	extAprSw					:BOOL:=FALSE;//气缸伸出感应器信号,需要链接到实际的IO点
	retAprSw					:BOOL:=FALSE;//气缸收回感应器信号,需要链接到实际的IO点
	enableExtAprSw				:BOOL:=TRUE;//启用伸出感应器,针对只有一个传感器的气缸
	enableRetAprSw				:BOOL:=TRUE;//启用收回感应器,针对只有一个传感器的气缸
	noteWTXT_Ext				:WSTRING(255):="";//气缸伸出动作NoteTXT 中文
	noteWTXT_Ret				:WSTRING(255):="";//气缸缩回动作NoteTXT 中文
END_VAR
VAR_OUTPUT
	extRelay				:BOOL:=FALSE;//气缸伸出执行继电器,需要链接到实际的IO点
	retRelay				:BOOL:=FALSE;//气缸收回执行继电器,需要链接到实际的IO点
	note_Ext				:BOOL:=FALSE;// 操作提示：true 伸出、打开执行无法下发
	note_Ret				:BOOL:=FALSE;// 操作提示：true 缩回、关闭执行无法下发
	busy					:BOOL;//气缸动作Busy状态
	done					:BOOL;//气缸动作Done状态
	extdone					:BOOL;//气缸动作伸出完成
	retdone					:BOOL;//气缸动作收回完成
	error					:BOOL;//气缸动作error状态
	errID					:UDINT;//气缸动作errID
	errTXT					:STRING(255):='';//气缸动作errTXT
	errWTXT					:WSTRING(255):="";//气缸动作errTXT 中文
	sensorShow				:STRING;
END_VAR
	
VAR
	firstPower:BOOL:=TRUE;
	extErrorDelayTon		:Ton;
	extDoneDelayTon			:Ton;
	retErrorDelayTon		:Ton;
	retDoneDelayTon			:Ton;
	
	extendTrigRAlc			:R_Trig;//上升沿触发
	
	singleControlR			:R_Trig;//上升沿触发
	singleControlF			:F_Trig;//上升沿触发
	
	extendTrigR1			:R_Trig;//上升沿触发
	retractTrigR1			:R_Trig;//上升沿触发
	resetTrigR1				:R_Trig;//上升沿触发
	stopTrigR1				:R_Trig;//上升沿触发
	powerTrigR1				:R_Trig;//上升沿触发
	
	errorStep				:UINT:=0;
	
	notBusyMonitorDelayTon:TON;//动作不切换时，延迟检测
	notBusyMonitorDelayTime:TIME:=T#2S;//动作不切换延迟检测时间
	noteTON_P:tON;            // 操作提示标志位延时继电器
	noteTON_N:tON;            // 操作提示标志位延时继电器
	noteRTrig_P:R_TRIG;          // 操作提示
	noteRTrig_N:R_TRIG;          // 操作提示
	extcheckDelayTime	:TON; // 输出到输入检测时间
	extcheckDelayTimeS	:TIME; // 输出到输入检测时间
	extcheckRtrig:R_TRIG;     // 输出到输入检测
	retcheckDelayTime	:TON; // 输出到输入检测时间
	retcheckDelayTimeS	:TIME; // 输出到输入检测时间
	retcheckRtrig:R_TRIG;     // 输出到输入检测
	extRealayRtrig:R_TRIG;
	retRealayRtrig:R_TRIG;
END_VAR

// 实时读取设置的流量值以及实际反馈浏览值
// ****************************
Init_ACT();
Error_ACT();
Extend_ACT();
Retract_ACT();
Reset_ACT();
Error_ACT();
SafeMonitor_ACT();
//首次上电，传感器状态决定电磁阀输出信号
//IF NOT firstPower THEN
//	IF extAprSw AND NOT retAprSw THEN
//		extend:=TRUE;
//		firstPower:=TRUE;
//	END_IF
//	IF retAprSw AND NOT extAprSw THEN
//		retract:=TRUE;
//		firstPower:=TRUE;
//	END_IF
//	IF (NOT extAprSw) AND (NOT retAprSw) THEN
//		errorStep:=3;
//	END_IF
//	IF (extAprSw) AND (retAprSw) THEN
//		errorStep:=3;
//	END_IF
//END_IF

(*
触发伸出动作，成功触发返回TRUE，触发失败返回FALSE
*)
METHOD Act_Extend : BOOL
VAR_INPUT
END_VAR
IF enable AND extCondition THEN// AND NOT busy
	Act_Extend:=extend:=TRUE;
ELSE
	Act_Extend:=FALSE;
END_IF
END_METHOD

(*
触发复位报警动作，成功触发返回TRUE，触发失败返回FALSE
*)
METHOD Act_Reset : BOOL
VAR_INPUT
END_VAR
Act_Reset:=reset:=TRUE;
END_METHOD

(*
触发缩回动作，成功触发返回TRUE，触发失败返回FALSE
*)
METHOD Act_Retract : BOOL
VAR_INPUT
END_VAR
IF enable AND retCondition THEN// AND NOT busy
	Act_Retract:=retract:=TRUE;
ELSE
	Act_Retract:=FALSE;
END_IF
END_METHOD

(*
触发停止输出动作，成功触发返回TRUE，触发失败返回FALSE
*)
METHOD Act_Stop : BOOL
VAR_INPUT
END_VAR
Act_Stop:=stop:=TRUE;
END_METHOD

ACTION Error_ACT:
CASE errorStep OF
	0:
		error:=FALSE;
		errID:=0;
		errTXT:='';
 (*
	1:
		error:=TRUE;
		errID:=errorID+errorStep;
		errTXT:=CONCAT(STR1:=nameTXT,STR2:=' Extend Error!');
		errWTXT:=WCONCAT(STR1:=TO_WSTRING(nameTXT),STR2:=" 伸出(打开)错误");
	2:
		error:=TRUE;
		errID:=errorID+errorStep;
		errTXT:=CONCAT(STR1:=nameTXT,STR2:=' Retract Error!');
		errWTXT:=WCONCAT(STR1:=TO_WSTRING(nameTXT),STR2:=" 缩回(关闭)错误");
		*)
	1..3:
		error:=TRUE;
		errID:=getErrID(errorStep);
		errTXT:=getErrTXT(errorStep);
		errWTXT:=getErrWTXT(errorStep);
END_CASE
END_ACTION

ACTION Extend_ACT:
//气缸伸出--extend 触发
IF extend AND NOT extCondition THEN
	note_Ext:=TRUE;
	note_Ret:=FALSE;
	NoteHMI.showFlag:=TRUE;
	NoteHMI.showText:='';
	NoteHMI.showText:=CONCAT(NoteHMI.showText,nameTXT);
	NoteHMI.showText:=CONCAT(NoteHMI.showText,' Ext Condition Not Satisfied!');
	operatorLog.append(CONCAT(nameTXT,' Extend Not Done'));
END_IF
IF extend AND enable AND extCondition THEN// AND NOT busy
	busy:=TRUE;
	retract:=FALSE;
	extdone:=FALSE;
	retdone:=FALSE;
	extStep:=10;
	retStep:=0;
	note_Ext:=FALSE;
	note_Ret:=FALSE;
	operatorLog.append(CONCAT(nameTXT,' Extend Done'));
	//errorStep:=0;
END_IF
extend:=FALSE;
extcheckDelayTime(IN:=extStep>10 AND NOT extcheckRtrig.Q,PT:=T#60S);
extcheckRtrig(CLK:=extAprSw);
IF extcheckRtrig.Q THEN
	extcheckDelayTimeS:=extcheckDelayTime.ET;
END_IF
CASE extStep OF
0:
	//ready
10:
	firstPower:=FALSE;
	extErrorDelayTon(IN:=FALSE);
	extDoneDelayTon(IN:=FALSE);
	extStep:=20;
	extRelay:=TRUE;
	retRelay:=FALSE;
20:
	extErrorDelayTon(IN:=(NOT extAprSw AND enableExtAprSw),PT:=errorDelayTime);
	IF extErrorDelayTon.Q THEN
		//done:=FALSE;
		extdone:=FALSE;
		retdone:=FALSE;
		errorStep:=1;
		RETURN;
	END_IF
	IF enableExtAprSw THEN
		extDoneDelayTon(IN:=extAprSw,PT:=doneDelayTimeShortExtend);
	ELSE
		extDoneDelayTon(IN:=NOT enableExtAprSw,PT:=doneDelayTimeLongExtend);
	END_IF
	
	IF extDoneDelayTon.Q THEN
		IF NOT retAprSw THEN
			busy:=FALSE;
			//done:=TRUE;
			extdone:=TRUE;
			retdone:=FALSE;
			errorStep:=0;
			IF NOT power AND NOT (CylinderType_Vacuum=cylinderType) THEN
				extRelay:=FALSE;
				retRelay:=FALSE;
			END_IF
		ELSE
			busy:=FALSE;
			//done:=TRUE;
			extdone:=FALSE;
			retdone:=FALSE;
			errorStep:=1;
		END_IF
	END_IF
END_CASE
END_ACTION

METHOD Get_Done_Ext : BOOL
VAR_INPUT
END_VAR
Get_Done_Ext:=extdone;
END_METHOD

METHOD Get_Done_Ret : BOOL
VAR_INPUT
END_VAR
Get_Done_Ret:=retdone;
END_METHOD

METHOD getErrID : UDINT
VAR_INPUT
	errID					:UDINT;//取值范围1~2
END_VAR
VAR
	nErrID					:UDINT;
END_VAR
nErrID:=errorID+errID;

getErrID:=nErrID;
END_METHOD

METHOD getErrTXT : STRING(255)
VAR_INPUT
	errID					:UDINT;//取值范围1~2
END_VAR
VAR
	sErrTXT					:STRING(255);
END_VAR

CASE errID OF
	1:
		sErrTXT:=CONCAT(STR1:=nameTXT,STR2:=' Extend Error!');
	2:
		sErrTXT:=CONCAT(STR1:=nameTXT,STR2:=' Retract Error!');
	3:
		sErrTXT:=CONCAT(STR1:=nameTXT,STR2:=' SensorCheck Error!');
ELSE
	sErrTXT:=CONCAT(STR1:=nameTXT,STR2:='');
END_CASE
getErrTXT:=sErrTXT;
END_METHOD

METHOD getErrWTXT : WSTRING(255)
VAR_INPUT
	errID					:UDINT;//取值范围1~16
END_VAR
VAR
	sErrTXT					:WSTRING(255);
END_VAR

CASE errID OF
	1:
		sErrTXT:=WCONCAT(STR1:=TO_WSTRING(nameTXT),STR2:=" 伸出(打开)错误");
	2:
		sErrTXT:=WCONCAT(STR1:=TO_WSTRING(nameTXT),STR2:=" 缩回(关闭)错误");
	3:
		sErrTXT:=WCONCAT(STR1:=TO_WSTRING(nameTXT),STR2:=" 传感器检测异常");
ELSE
	sErrTXT:=WCONCAT(STR1:=TO_WSTRING(nameTXT),STR2:="");
END_CASE
getErrWTXT:=sErrTXT;
END_METHOD

ACTION Init_ACT:
done:=(extdone OR retdone);
InitHMI_ACT();
manualCtrl_ACT();


noteTON_P(IN:=note_Ext,PT:=T#0.1S);
noteRTrig_P(CLK:=noteTON_P.Q);
IF noteRTrig_P.Q THEN
//	gLog_Note.append_EX(noteWTXT_Ext);
END_IF
noteTON_N(IN:=note_Ret,PT:=T#0.1S);
noteRTrig_N(CLK:=noteTON_N.Q);
IF noteRTrig_N.Q THEN
//	gLog_Note.append_EX(noteWTXT_Ret);
END_IF
extRealayRtrig(CLK:=extRelay);
IF extRealayRtrig.Q THEN
	HMIItf.singleControl:=TRUE;
END_IF
retRealayRtrig(CLK:=NOT extRelay);
IF retRealayRtrig.Q THEN
	HMIItf.singleControl:=FALSE;
END_IF
END_ACTION

ACTION InitHMI_ACT:
HMIItf.extAprSw:=extAprSw;
HMIItf.retAprSw:=retAprSw;
HMIItf.enableExt:=enableExtAprSw;
HMIItf.enableRet:=enableRetAprSw;
HMIItf.HMIEnable:=hmiEN;
HMIItf.enable:=enable;
HMIItf.done:=done;
HMIItf.busy:=busy;
HMIItf.error:=error;
HMIItf.errID:=UDINT_TO_DINT(errID);
HMIItf.errTXT:=errTXT;
HMIItf.extRelay:=extRelay;
HMIItf.retRelay:=retRelay;
HMIItf.power:=power;
HMIItf.nameTXT:=nameTXT;
HMIItf.extenderror:=error AND errorID=1;
HMIItf.retracterror:=error AND errorID=2;
HMIItf.extcondition:=extCondition;
HMIItf.retcondition:=retCondition;
HMIItf.sensorShow:=sensorShow;
END_ACTION

ACTION ManualCtrl_ACT:
//HMI手动控制
//IF ctrlMode=eManualCtrMode THEN
IF hmiEN THEN
	extendTrigRAlc(CLK:=HMIItf.extendAndretract);
	IF extendTrigRAlc.Q THEN// AND NOT busy
		IF extRelay THEN//如果伸出继电器或伸出传感器亮，则认为已经伸出过
			retract:=TRUE;
		END_IF
		IF retRelay THEN
			extend:=TRUE;
		END_IF
		IF NOT extRelay AND NOT retRelay THEN
			IF extAprSw THEN
				retract:=TRUE;
			END_IF
			IF retAprSw THEN
				extend:=TRUE;
			END_IF
		END_IF
	END_IF
	singleControlR(CLK:=HMIItf.singleControltemp);
	extendTrigR1(CLK:=HMIItf.extend );
	IF extendTrigR1.Q OR (singleControlR.Q AND NOT HMIItf.singleControl) THEN// AND NOT busy
		HMIItf.extend:=FALSE;
		WarmHMI.showText:='';
		WarmHMI.showFlag:=TRUE;
		WarmHMI.showText:=CONCAT(WarmHMI.showText,'Are you sure you want to Extend the ');
		WarmHMI.showText:=CONCAT(WarmHMI.showText,nameTXT);
		WarmHMI.showText:=CONCAT(WarmHMI.showText,' ?');
	END_IF
	IF WarmHMI.bOK AND NOT WarmHMI.showFlag AND FIND(WarmHMI.showText,nameTXT)>0 AND FIND(WarmHMI.showText,'Extend')>0 THEN
		extend:=TRUE;
		HMIItf.extend:=FALSE;
		IF HMIItf.singleControl THEN
			;
		ELSE
			IF extCondition THEN
				HMIItf.singleControl:=TRUE;
			END_IF
		END_IF
		WarmHMI.bOK:=FALSE;
		WarmHMI.showText:='';
	END_IF
	IF WarmHMI.bNO AND NOT WarmHMI.showFlag AND FIND(WarmHMI.showText,nameTXT)>0 AND FIND(WarmHMI.showText,'Extend')>0 THEN
		HMIItf.extend:=FALSE;
		WarmHMI.bNO:=FALSE;
		WarmHMI.showText:='';
	END_IF
	
	retractTrigR1(CLK:=HMIItf.retract);
	IF retractTrigR1.Q OR (singleControlR.Q AND HMIItf.singleControl) THEN// AND NOT busy
		HMIItf.retract:=FALSE;
		WarmHMI.showText:='';
		WarmHMI.showFlag:=TRUE;
		WarmHMI.showText:=CONCAT(WarmHMI.showText,'Are you sure you want to Retract the ');
		WarmHMI.showText:=CONCAT(WarmHMI.showText,nameTXT);
		WarmHMI.showText:=CONCAT(WarmHMI.showText,' ?');
	END_IF
	IF WarmHMI.bOK AND NOT WarmHMI.showFlag AND FIND(WarmHMI.showText,nameTXT)>0 AND FIND(WarmHMI.showText,'Retract')>0 THEN
		retract:=TRUE;
		HMIItf.retract:=FALSE;
		IF HMIItf.singleControl  THEN
			IF retCondition THEN
				HMIItf.singleControl:=FALSE;
			END_IF
		ELSE
			;
		END_IF
		WarmHMI.bOK:=FALSE;
		WarmHMI.showText:='';
	END_IF
	IF WarmHMI.bNO AND NOT WarmHMI.showFlag AND FIND(WarmHMI.showText,nameTXT)>0 AND FIND(WarmHMI.showText,'Retract')>0 THEN
		WarmHMI.bNO:=FALSE;
		HMIItf.retract:=FALSE;
		WarmHMI.showText:='';
	END_IF
	
	stopTrigR1(CLK:=HMIItf.stop);
	IF stopTrigR1.Q THEN// AND NOT busy
		stop:=TRUE;
	END_IF
	
	powerTrigR1(CLK:=HMIItf.power);
	IF powerTrigR1.Q THEN// AND NOT busy
		IF power THEN
			power:=FALSE;
		ELSE
			power:=TRUE;
		END_IF
	END_IF
END_IF
IF extAprSw THEN
	sensorShow:='UP';
ELSIF retAprSw THEN
	sensorShow:='DOWN';
ELSE
	sensorShow:='<->';
END_IF
END_ACTION

ACTION Reset_ACT:
IF reset THEN
	IF NOT power THEN
		extRelay:=FALSE;
		retRelay:=FALSE;
	END_IF
	busy:=FALSE;
	//done:=FALSE;
	//extdone:=FALSE;
	//retdone:=FALSE;
	errorStep:=0;
	note_Ext:=FALSE;
	note_Ret:=FALSE;
	reset:=FALSE;
END_IF

IF stop THEN
	stop:=FALSE;
	extRelay:=FALSE;
	retRelay:=FALSE;
	note_Ext:=FALSE;
	note_Ret:=FALSE;
	//无自锁检测说法，直接停
//	extStep:=0;
//	retStep:=0;
END_IF
END_ACTION

ACTION Retract_ACT:
//气缸收回--retract 触发
IF retract AND NOT retCondition THEN
	note_Ret:=TRUE;
	note_Ext:=FALSE;
	NoteHMI.showFlag:=TRUE;
	NoteHMI.showText:='';
	NoteHMI.showText:=CONCAT(NoteHMI.showText,nameTXT);
	NoteHMI.showText:=CONCAT(NoteHMI.showText,' Ret Condition Not Satisfied!');
	operatorLog.append(CONCAT(nameTXT,' Retract Not Done'));
END_IF
IF retract AND enable AND retCondition THEN// AND NOT busy
	busy:=TRUE;
	extend:=FALSE;
	extdone:=FALSE;
	retdone:=FALSE;
	extStep:=0;
	retStep:=10;
	note_Ext:=FALSE;
	note_Ret:=FALSE;
	operatorLog.append(CONCAT(nameTXT,' Retract Done'));
	//errorStep:=0;
END_IF
retract:=FALSE;
retcheckDelayTime(IN:=retStep>10 AND NOT retcheckRtrig.Q,PT:=T#60S);
retcheckRtrig(CLK:=retAprSw);
IF retcheckRtrig.Q THEN
	retcheckDelayTimeS:=retcheckDelayTime.ET;
END_IF
CASE retStep OF
0:
	//ready
	
10:
	firstPower:=FALSE;
	retErrorDelayTon(IN:=FALSE);
	retDoneDelayTon(IN:=FALSE);
	retStep:=20;
	extRelay:=FALSE;
	viewForlineVac:=inVacu;
	retRelay:=TRUE;
20:
	retErrorDelayTon(IN:=(NOT retAprSw AND enableRetAprSw),PT:=errorDelayTime);
	IF retErrorDelayTon.Q THEN
		//done:=FALSE;
		extdone:=FALSE;
		retdone:=FALSE;
		errorStep:=2;
		RETURN;
	END_IF
	IF enableRetAprSw THEN
		retDoneDelayTon(IN:=retAprSw,PT:=doneDelayTimeShortRetract);
	ELSE
		retDoneDelayTon(IN:=NOT enableRetAprSw,PT:=doneDelayTimeLongRetract);
	END_IF
	
	IF retDoneDelayTon.Q THEN
		IF NOT extAprSw THEN
			busy:=FALSE;
			//done:=TRUE;
			extdone:=FALSE;
			retdone:=TRUE;
			errorStep:=0;
			IF NOT power AND NOT (CylinderType_Vacuum=cylinderType) THEN
				extRelay:=FALSE;
				retRelay:=FALSE;
			END_IF
			IF CylinderType_Vacuum=cylinderType THEN
				retRelay:=FALSE;
			END_IF
		ELSE
			busy:=FALSE;
			//done:=TRUE;
			extdone:=FALSE;
			retdone:=FALSE;
			errorStep:=2;
		END_IF
	END_IF
END_CASE
END_ACTION

ACTION SafeMonitor_ACT:
notBusyMonitorDelayTon(IN:=NOT busy,PT:=notBusyMonitorDelayTime);
IF real_TimeMonitor THEN
	IF notBusyMonitorDelayTon.Q THEN
		//伸出实时检测
		IF (enableExtAprSw AND NOT extAprSw) AND extRelay THEN
			errorStep:=1;
		END_IF
	
		//缩回实时检测	
		IF (enableRetAprSw AND NOT retAprSw) AND retRelay  THEN
			errorStep:=2;
		END_IF
//		IF cylinderType=CylinderType_ButV THEN
//			IF NOT extCondition AND (NOT retdone OR extRelay) AND NOT firstPower THEN//蝶阀单控，检测到开条件消失，强制关闭
//				errorStep:=1;
//				extRelay:=FALSE;
//				retract:=TRUE;
//				firstPower:=FALSE;
//			END_IF
//		END_IF
		IF firstPower THEN
			firstPower:=FALSE;
			IF extAprSw THEN
				HMIItf.singleControl:=TRUE;
			END_IF
			IF retAprSw THEN
				HMIItf.singleControl:=FALSE;
			END_IF
		END_IF
	END_IF
END_IF
END_ACTION

ACTION VersionLog:
(*
版本: V1.0.0.0
说明:
	1. 首个版本
	2. 含普通气缸\真空吸类型的控制
	3. 可配置是否有到位信号, 以及到位稳定时间
(--------------------------------------------------)
新版本: V1.0.1.0
更新时间: 2019/11/20 19:00
更新说明:
	1. 优化编写方式
	2. 修改错误编码起始位，现改为从1开始
(--------------------------------------------------)
新版本: V1.0.1.1
更新时间: 2020/03/23 23:00
更新说明:
	1. 优化报错方式
	2. 增加伸出、缩回、复位和停止触发函数
(--------------------------------------------------)
新版本: V1.0.1.2
更新时间: 2020/04/22 09:50
更新说明:
	1. 增加中文报警输出
(--------------------------------------------------)
新版本: V1.0.1.3
更新时间: 2020/09/16
更新说明:
	1. 开放错误ID、错误文本信息获取接口
(--------------------------------------------------)
新版本: V1.0.1.4
更新时间: 2020/10/06
更新说明:
	1. 移除控制模式变量，增加HMI启用条件
	2. 增加外部获取伸出缩回完成信号接口函数
(--------------------------------------------------)
新版本: V1.0.1.5
更新时间: 2020/10/14
更新说明:
	1. 优化代码
(--------------------------------------------------)
*)
END_ACTION

END_FUNCTION_BLOCK

// ---- POUs/BaseModule/PrintLogModule_EX/printLogModule_EX.TcPOU
FUNCTION_BLOCK printLogModule_EX
VAR_INPUT
	sRootDirPath	:T_MaxString:='C:\Log';//根目录
	sFileName		:T_MaxString:='log.txt';//Log文件名
	enable			:BOOL:=FALSE;//是否启用Log保存到文件功能
	enableShowInfo	:BOOL:=TRUE;//是否启用ShowInfo功能---HMI
	clearShowInfo	:BOOL:=FALSE;//清除HMI显示
	
	enableDelete	:BOOL;
	storageDays		:UINT:=7;
	sAmsNetId		:STRING;//获取arrAmsNetId
END_VAR
VAR_OUTPUT
	busy			:BOOL:=FALSE;
	error			:BOOL:=FALSE;
	errID			:UDINT:=0;
	errTxt			:STRING(255):='';
END_VAR
VAR
	strData			:ARRAY [cNumBegin..(cNumLength+cNumBegin-1)] OF printLogModule_EX_DataST;
	length			:DINT:=0;
	endPoint		:DINT:=cNumBegin;
	//popup
	popupStep		:UINT:=0;
	popupTON		:TON;
	//Save Log
	saveStep		:UINT:=0;
	saveStr			:WSTRING(255);//保存的信息
	saveStrBuff		:WSTRING(255);//保存的信息-buffer
	{ attribute 'TcEncoding' := 'UTF-8'}
	saveStrBuff1	:STRING(255);//保存的信息-buffer
	saveB			:BOOL:=FALSE;//触发保存
	sBusy			:BOOL:=FALSE;
	sDone			:BOOL:=FALSE;
	//ShowInfo
	HMIData						:printLogModule_EX_DataHMI;
	clearShowInfoR1				:R_Trig;
	iClearTemp					:DINT;
	enableSaveR_Trig			:R_Trig;
	enableSaveF_Trig			:F_Trig;
	enableSaveShowLogR_Trig		:R_Trig;
	
//File
	hFile			: UINT:= 0;(* File handle of the source file *)
	fbCreateDir		: FB_CreateDir;//Creat File
	fbFileOpen		: FB_FileOpen;//Creat file.if file didn't exist, then creat it.
	//fbFileGets	: FB_FileGets;//
	//fbFilePuts		: FB_FilePuts;//
	fbFileWrite		: FB_FileWrite;//  
	fbFileClose		: FB_FileClose;//Close File
	
	sChildDirPath1	: T_MaxString:='';//子目录
	sChildDirName1	: T_MaxString:='';//子文件夹名
	sFilePathName	: T_MaxString:='';//Log文件路径
	(* Save show log *)
	saveShowLogStep			:UINT:=0;
	saveShowLogStr			:WSTRING(255);// ShowLog 保存的信息
	saveShowLogStrBuff		:WSTRING(255);// ShowLog 保存的信息-buffer
	saveShowLogStrBuff1		:STRING(255);// ShowLog 保存的信息-buffer
	saveShowLogB			:BOOL:=FALSE;// ShowLog 触发保存
	bShowLogBusy			:BOOL:=FALSE;// ShowLog busy
	sShowLogDone			:BOOL:=FALSE;// ShowLog done
	
	hShowLogFile			: UINT:= 0;(* ShowLog File handle of the source file *)
	fbShowLogCreateDir		: FB_CreateDir;// ShowLog Creat File
	fbShowLogFileOpen		: FB_FileOpen;// ShowLog Creat file.if file didn't exist, then creat it.
	fbShowLogFileWrite		: FB_FileWrite;// ShowLog 
	fbShowLogFileClose		: FB_FileClose;// ShowLog Close File
	
	sShowLogChildDirPath1	: T_MaxString:='';// ShowLog 子目录
	sShowLogChildDirName1	: T_MaxString:='';// ShowLog 子文件夹名
	sShowLogFilePathName	: T_MaxString:='';// ShowLog Log文件路径
	
	iShowLogTemp			:DINT:=0;
	showLogStrData			:ARRAY [cNumBegin_showInof..cNumLength_showInof] OF printLogModule_EX_DataST;
//获取系统时间
	ntGetTime				: NT_GetTime;
	systemTimeStruct		: TIMESTRUCT;
	getSystemTimeStep		: UINT:=0;
	systemTIMEStr			: STRING:='';//系统时间，格式YYYY-MM-DD hh:mm:ss_zzz
	sysTIMEStrYY			: STRING:='';//系统时间，年
	sysTIMEStrMM			: STRING:='';//系统时间，月
	sysTIMEStrDD			: STRING:='';//系统时间，日
	sysTIMEStr_HH			: STRING:='';//系统时间，时
	sysTIMEStr_mm			: STRING:='';//系统时间，分
	sysTIMEStr_ss			: STRING:='';//系统时间，秒
	//popup
	iTempPopup				:DINT;
	_leng					:DINT;
	//detele file
	detele_file_step		:UINT:=0;
	delete_index			:UINT;
	delete_index_temp		:UINT;
	fbFileDelete			:FB_FileDelete;
	fbRemoveDir				:FB_RemoveDir;
	delete_done				:BOOL;
END_VAR
VAR PERSISTENT
	//delete file
	deletePathTemp			:STRING;
	stDeleteFile			:ARRAY [1..35] OF ST_DeleteFile;
END_VAR
VAR
	bWrtie					: BOOL;//触发断电保持保存
	//fbUPS					: FB_S_UPS;
	fbUPS					: FB_S_UPS_CX51x0;
	fbGetCurTaskIndex		: GetCurTaskIndex;
	fbWritePersistentData	: FB_WritePersistentData;
	nTaskNo					: INT;
	wrtieR_TRIG				: R_TRIG;
END_VAR

(*
旧版本: V1.0.0.0
新版本: V1.0.0.1
更新时间: 2019/07/09 10:30
更新说明:
	1. 更新文件保存格式, 时间和内容改为逗号分隔
	2. 修改每个保存内容后缀为$N
*)
getSystemTime(sAmsNetId);
popup();
saveLog();
saveShowLog();
deleteFile();
WPersData();//执行断电保持处理

clearShowInfoR1(CLK:=clearShowInfo OR HMIData.clearInformation);
IF clearShowInfoR1.Q THEN
	FOR iClearTemp:=cNumBegin_showInof TO cNumLength_showInof BY 1 DO
		HMIData.logStrData[iClearTemp].sTime:="";
		HMIData.logStrData[iClearTemp].msg:="";
	END_FOR
END_IF
enableSaveR_Trig(CLK:=HMIData.enableSave);
IF enableSaveR_Trig.Q THEN
	enable:=TRUE;
END_IF
enableSaveF_Trig(CLK:=HMIData.enableSave);
IF enableSaveF_Trig.Q THEN
	enable:=FALSE;
END_IF
HMIData.enableSave:=enable;

enableSaveShowLogR_Trig(CLK:=HMIData.enableSaveShowLog AND NOT bShowLogBusy);
IF enableSaveShowLogR_Trig.Q THEN
	saveShowLogB:=TRUE;
END_IF

METHOD appedFree : BOOL
VAR_INPUT
	languageFlag:BOOL;
	str:STRING;
	wstr:WSTRING;
END_VAR
IF languageFlag THEN
	append(str);
ELSE
	append_EX(wstr);
END_IF
appedFree:=TRUE;
END_METHOD

//只能添加 英文 字符数据
METHOD append : BOOL
VAR_INPUT
	{ attribute 'TcEncoding' := 'UTF-8'}
	str		:T_MaxString;
END_VAR
append_EX(TO_WSTRING(str));
END_METHOD

//可添加 中文 字符数据
METHOD append_EX : BOOL
VAR_INPUT
	str		:WSTRING(255);
END_VAR
VAR
	sTime	:WSTRING(255);
END_VAR
busy:=TRUE;

sTime:=TO_WSTRING(systemTIMEStr);
//str:=CONCAT(STR1:=CONCAT(STR1:=systemTIMEStr,STR2:=': '),STR2:=str);
IF enableShowInfo THEN
	showInfo(sTime:=sTime, str:=str);
END_IF
str:=WCONCAT(STR1:=str,STR2:="$N");//'$R$N'
IF endPoint>=(cNumLength-1) THEN
	busy:=FALSE;
	RETURN;
END_IF
strData[endPoint].sTime:=sTime;
strData[endPoint].msg:=str;
endPoint:=endPoint+1;
length:=endPoint-cNumBegin;

busy:=FALSE;
END_METHOD

METHOD PRIVATE deleteFile
VAR_INPUT
END_VAR
fbFileDelete(
	sNetId:= , 
	sPathName:= , 
	ePath:= , 
	bExecute:= , 
	tTimeout:= , 
	bBusy=> , 
	bError=> , 
	nErrId=> );
fbRemoveDir(
	sNetId:= , 
	sPathName:= , 
	ePath:= , 
	bExecute:= , 
	tTimeout:= , 
	bBusy=> , 
	bError=> , 
	nErrId=> );
CASE detele_file_step OF
	0:
		IF enableDelete AND NOT delete_done THEN
			detele_file_step:=10;
		END_IF
	10:
		delete_index_temp:=storageDays+1;
		IF storageDays<=0 THEN
			delete_index_temp:=1+1;
		ELSIF storageDays>=30 THEN
			delete_index_temp:=30+1;
		END_IF
		
		detele_file_step:=detele_file_step+10;
	20:
		fbFileDelete(
			bExecute:= FALSE, );
		detele_file_step:=detele_file_step+10;
	30:
		detele_file_step:=detele_file_step+10;
	40:
		fbFileDelete(
			sPathName:= stDeleteFile[delete_index_temp].sFilePath, 
			bExecute:= TRUE, );
		IF fbFileDelete.bBusy THEN
			detele_file_step:=detele_file_step+10;
		END_IF
	50:
		IF NOT fbFileDelete.bBusy OR fbFileDelete.bError THEN
			delete_index_temp:=delete_index_temp+1;
			IF delete_index_temp>35 THEN
				detele_file_step:=60;
			ELSE
				detele_file_step:=20;
			END_IF
		END_IF
	60:
		fbFileDelete(
			bExecute:= FALSE, );
		delete_done:=TRUE;
		detele_file_step:=0;
END_CASE
END_METHOD

METHOD PRIVATE getSystemTime : BOOL
VAR_INPUT
	systemId		:STRING;
END_VAR
//获取本地系统时间--输出到变量 systemTIMEStr
CASE getSystemTimeStep OF
0:
	ntGetTime(
		NETID:= systemId , 
		START:= FALSE, 
		TMOUT:= , 
		BUSY=> , 
		ERR=> , 
		ERRID=> , 
		TIMESTR=> systemTimeStruct);
	IF NOT ntGetTime.BUSY AND NOT ntGetTime.ERR THEN
		getSystemTimeStep:=getSystemTimeStep+1;
	END_IF
1:
	ntGetTime(
		NETID:=systemId , 
		START:= TRUE, 
		TMOUT:= , 
		BUSY=> , 
		ERR=> , 
		ERRID=> , 
		TIMESTR=> systemTimeStruct);
	IF NOT ntGetTime.BUSY AND NOT ntGetTime.ERR THEN
		systemTIMEStr:=SYSTEMTIME_TO_STRING(systemTimeStruct);//系统时间转成字符串格式
		
		sysTIMEStrYY:=WORD_TO_DECSTR(in:=systemTimeStruct.wYear,iPrecision:=4);
		sysTIMEStrMM:=WORD_TO_DECSTR(in:=systemTimeStruct.wMonth,iPrecision:=2);
		sysTIMEStrDD:=WORD_TO_DECSTR(in:=systemTimeStruct.wDay,iPrecision:=2);
		sysTIMEStr_HH:=WORD_TO_DECSTR(in:=systemTimeStruct.wHour,iPrecision:=2);
		sysTIMEStr_mm:=WORD_TO_DECSTR(in:=systemTimeStruct.wMinute,iPrecision:=2);
		sysTIMEStr_ss:=WORD_TO_DECSTR(in:=systemTimeStruct.wSecond,iPrecision:=2);
		sChildDirName1:=CONCAT(STR1:=CONCAT(STR1:=sysTIMEStrYY,STR2:=sysTIMEStrMM),STR2:=sysTIMEStrDD);
		sShowLogChildDirName1:=CONCAT(STR1:=CONCAT(STR1:=sysTIMEStrYY,STR2:=sysTIMEStrMM),STR2:=sysTIMEStrDD);
		
		deletePathTemp:=CONCAT(CONCAT(sRootDirPath,'\'), sChildDirName1);
		IF deletePathTemp<>stDeleteFile[1].sDirPath THEN
			FOR delete_index:=35 TO 2 BY -1 DO
				stDeleteFile[delete_index]:=stDeleteFile[delete_index-1];
				stDeleteFile[delete_index].nCount:=delete_index;
			END_FOR
			stDeleteFile[1].sDirPath:=deletePathTemp;
			stDeleteFile[1].sFilePath:=CONCAT(CONCAT(deletePathTemp,'\'),sFileName);
			stDeleteFile[1].nCount:=1;
			delete_done:=FALSE;
			bWrtie:=TRUE;
			WPersData();//执行断电保持处理
		END_IF
		
		getSystemTimeStep:=0;
	ELSIF ntGetTime.ERR THEN
		systemTIMEStr:='';
		getSystemTimeStep:=0;
	END_IF	
END_CASE
END_METHOD

METHOD PRIVATE popup : BOOL
VAR_INPUT
END_VAR
CASE popupStep OF
0:
	IF length>0 AND NOT busy AND NOT sBusy THEN
		_leng:=length;
		//saveStr:=strData[cNumBegin];
		saveStr:=WCONCAT(WCONCAT(strData[cNumBegin].sTime,","),strData[cNumBegin].msg);
		FOR iTempPopup:=cNumBegin TO (_leng-1) DO
			strData[iTempPopup]:=strData[iTempPopup+1];
		END_FOR
		endPoint:=endPoint-1;
		length:=endPoint-cNumBegin;
		popupStep:=10;
		saveB:=TRUE;
	END_IF
	
10:
	IF sBusy OR NOT enable THEN
		popupStep:=11;
	END_IF
11:
	IF NOT sBusy OR NOT enable THEN
		popupStep:=12;
	END_IF
	popupTON(IN:=FALSE);
12:
	popupTON(IN:=NOT popupTON.Q,PT:=T#100MS);
	IF popupTON.Q THEN
		popupTON(IN:=FALSE);
		popupStep:=0;
	END_IF
END_CASE
END_METHOD

METHOD PRIVATE saveLog : BOOL
VAR_INPUT
END_VAR
//Log 保存
CASE saveStep OF
0:
	IF ''=sChildDirName1 THEN
		RETURN;
	END_IF
	IF saveB AND NOT sBusy AND enable THEN
		saveStrBuff:="";
		saveStrBuff:=saveStr;
		saveStr:="";
		
		saveStrBuff1:=WSTRING_TO_STRING(saveStrBuff);
		//STRING_TO_UTF8(ADR(saveStrBuff1),ADR(saveStrBuff1),SIZEOF(saveStrBuff1));
		WSTRING_TO_UTF8(ADR(saveStrBuff1),ADR(saveStrBuff),SIZEOF(saveStrBuff));
		
		sBusy:=TRUE;
		sDone:=FALSE;
		error:=FALSE;
		errID:=0;
		errTxt:='';
		
		sChildDirPath1:='';	
		sFilePathName:='';
		sChildDirPath1:=CONCAT(STR1:=CONCAT(STR1:=sRootDirPath,STR2:='\'),STR2:=sChildDirName1);
		sFilePathName:=CONCAT(STR1:=CONCAT(STR1:=sChildDirPath1,STR2:='\'),STR2:=sFileName);
		fbCreateDir(sNetId:= , bExecute:= FALSE);
		saveStep:=saveStep+1;
	END_IF
	saveB:=FALSE;
1:
	fbCreateDir(
			sNetId:= , 
			sPathName:= sRootDirPath, 
			ePath:= PATH_GENERIC, 
			bExecute:= TRUE, 
			tTimeout:= , 
			bBusy=> , 
			bError=> , 
			nErrId=> );
	IF NOT fbCreateDir.bBusy THEN
		fbCreateDir(
			sNetId:= , 
			bExecute:= FALSE);	
		saveStep:=saveStep+1;
	END_IF
2:
	fbCreateDir(
			sNetId:= , 
			sPathName:= sChildDirPath1, 
			ePath:= PATH_GENERIC, 
			bExecute:= TRUE, 
			tTimeout:= , 
			bBusy=> , 
			bError=> , 
			nErrId=> );
	IF NOT fbCreateDir.bBusy THEN
		fbCreateDir(
			sNetId:= , 
			bExecute:= FALSE);	
		saveStep:=saveStep+1;
	END_IF
3:
	fbFileOpen(
		sNetId:= , 
		sPathName:= sFilePathName, 
		nMode:= FOPEN_MODEAPPEND OR FOPEN_MODETEXT, 
		bExecute:= FALSE);
	saveStep:=saveStep+1;
4:
	fbFileOpen(
		sNetId:= , 
		sPathName:= sFilePathName, 
		nMode:= FOPEN_MODEAPPEND OR FOPEN_MODETEXT,
		ePath:= , 
		bExecute:= TRUE, 
		tTimeout:= , 
		bBusy=> , 
		bError=> , 
		nErrId=> , 
		hFile=> hFile);
	IF NOT fbFileOpen.bBusy THEN
		IF NOT fbFileOpen.bError THEN
			saveStep:=saveStep+1;
		ELSE
			saveStep:=50;//Error
		END_IF
	END_IF
5:
	fbFileWrite(
		sNetId:= , 
		hFile:= hFile, 
		pWriteBuff:= , 
		cbWriteLen:= , 
		bExecute:= FALSE, 
		tTimeout:= , 
		bBusy=> , 
		bError=> , 
		nErrId=> , 
		cbWrite=> );
	
	saveStep:=saveStep+1;
6:
	fbFileWrite(
		sNetId:= , 
		hFile:= hFile, 
		pWriteBuff:= ADR(saveStrBuff1), 
		cbWriteLen:= TO_UDINT(LEN(saveStrBuff1)), 
		bExecute:= TRUE, 
		tTimeout:= , 
		bBusy=> , 
		bError=> , 
		nErrId=> , 
		cbWrite=> );
	IF NOT fbFileWrite.bBusy AND NOT fbFileWrite.bError THEN
		saveStep:=30;
		fbFileClose(
			sNetId:= , 
			hFile:= hFile, 
			bExecute:= FALSE);
	ELSIF fbFileWrite.bError THEN
		saveStep:=50;
		fbFileClose(
			sNetId:= , 
			hFile:= hFile, 
			bExecute:= FALSE);
	END_IF

30:	//Done
	fbFileClose(
		sNetId:= , 
		hFile:= hFile, 
		bExecute:= TRUE, 
		tTimeout:= , 
		bBusy=> , 
		bError=> , 
		nErrId=> );
	IF NOT fbFileClose.bBusy THEN
		saveStep:=saveStep+1;
	END_IF
31:
	fbFileClose(
		sNetId:= , 
		hFile:= hFile, 
		bExecute:= FALSE);
	saveStep:=0;
	
	sBusy:=FALSE;
	sDone:=TRUE;
	error:=FALSE;
	errID:=0;
	errTxt:='';
	saveB:=FALSE;

50://Error
	fbFileClose(
		sNetId:= , 
		hFile:= hFile, 
		bExecute:= TRUE, 
		tTimeout:= , 
		bBusy=> , 
		bError=> , 
		nErrId=> );
	IF NOT fbFileClose.bBusy THEN
		saveStep:=saveStep+1;
	END_IF
51:
	fbFileClose(
		sNetId:= , 
		hFile:= hFile, 
		bExecute:= FALSE);
	saveStep:=0;
	
	sBusy:=FALSE;
	sDone:=FALSE;
	error:=TRUE;
	errID:=1;
	errTxt:='Log writing error!';
	saveB:=FALSE;
END_CASE
END_METHOD

METHOD PRIVATE saveShowLog : BOOL
VAR_INPUT
END_VAR
VAR
	bDataTemp:ARRAY [1..255] OF BYTE;
	pDstUTF8    : POINTER TO BYTE;;
END_VAR
//ShowLog 保存
CASE saveShowLogStep OF
0:
	IF ''=sShowLogChildDirName1 THEN
		RETURN;
	END_IF
	IF saveShowLogB AND NOT bShowLogBusy THEN
		showLogStrData:=HMIData.logStrData;
		
		bShowLogBusy:=TRUE;
		
		sShowLogChildDirPath1:='';	
		sShowLogFilePathName:='';
		sShowLogChildDirPath1:=CONCAT(STR1:=CONCAT(STR1:=sRootDirPath,STR2:='\'),STR2:=sShowLogChildDirName1);
		sShowLogFilePathName:=CONCAT(STR1:=CONCAT(STR1:=sShowLogChildDirPath1,STR2:='\'),
									 STR2:=CONCAT(STR1:=CONCAT(CONCAT(STR1:=CONCAT(STR1:=sysTIMEStrYY,STR2:=sysTIMEStrMM),STR2:=sysTIMEStrDD),
												  STR2:=CONCAT(STR1:=CONCAT(STR1:=sysTIMEStr_HH,STR2:=sysTIMEStr_mm),STR2:='')),sFileName));
		fbShowLogCreateDir(sNetId:= , bExecute:= FALSE);
		saveShowLogStep:=saveShowLogStep+1;
	END_IF
	saveShowLogB:=FALSE;
1:
	fbShowLogCreateDir(
			sNetId:= , 
			sPathName:= sRootDirPath, 
			ePath:= PATH_GENERIC, 
			bExecute:= TRUE, 
			tTimeout:= , 
			bBusy=> , 
			bError=> , 
			nErrId=> );
	IF NOT fbShowLogCreateDir.bBusy THEN
		fbShowLogCreateDir(
			sNetId:= , 
			bExecute:= FALSE);	
		saveShowLogStep:=saveShowLogStep+1;
	END_IF
2:
	fbShowLogCreateDir(
			sNetId:= , 
			sPathName:= sShowLogChildDirPath1, 
			ePath:= PATH_GENERIC, 
			bExecute:= TRUE, 
			tTimeout:= , 
			bBusy=> , 
			bError=> , 
			nErrId=> );
	IF NOT fbShowLogCreateDir.bBusy THEN
		fbShowLogCreateDir(
			sNetId:= , 
			bExecute:= FALSE);	
		saveShowLogStep:=saveShowLogStep+1;
	END_IF
3:
	fbShowLogFileOpen(
		sNetId:= , 
		sPathName:= sShowLogFilePathName, 
		nMode:= FOPEN_MODEWRITE OR FOPEN_MODETEXT, //FOPEN_MODEAPPEND OR FOPEN_MODETEXT, 
		bExecute:= FALSE);
	saveShowLogStep:=saveShowLogStep+1;
4:
	fbShowLogFileOpen(
		sNetId:= , 
		sPathName:= sShowLogFilePathName, 
		nMode:= FOPEN_MODEWRITE OR FOPEN_MODETEXT, //FOPEN_MODEAPPEND OR FOPEN_MODETEXT,   FOPEN_MODEBINARY
		ePath:= , 
		bExecute:= TRUE, 
		tTimeout:= , 
		bBusy=> , 
		bError=> , 
		nErrId=> , 
		hFile=> hShowLogFile);
	IF NOT fbShowLogFileOpen.bBusy THEN
		IF NOT fbShowLogFileOpen.bError THEN
			iShowLogTemp:=cNumBegin_showInof;
			saveShowLogStep:=50;
		ELSE
			saveShowLogStep:=500;//Error
		END_IF
	END_IF
50:
	IF iShowLogTemp<=cNumLength_showInof AND iShowLogTemp>=cNumBegin_showInof THEN
		IF ""<>showLogStrData[iShowLogTemp].sTime THEN
			//saveShowLogStr:=showLogStrData[iShowLogTemp];
			saveShowLogStr:=WCONCAT(WCONCAT(showLogStrData[iShowLogTemp].sTime,","),showLogStrData[iShowLogTemp].msg);
			saveShowLogStrBuff:="";
			saveShowLogStrBuff:=WCONCAT(saveShowLogStr,"$N");
			saveShowLogStr:="";
			
			saveShowLogStrBuff1:=WSTRING_TO_STRING(saveShowLogStrBuff);
			//STRING_TO_UTF8(ADR(saveShowLogStrBuff1),ADR(saveShowLogStrBuff1),SIZEOF(saveShowLogStrBuff1));
			//WSTRING_TO_UTF8(ADR(saveShowLogStrBuff),ADR(saveShowLogStrBuff),SIZEOF(saveShowLogStrBuff));
			saveShowLogStep:=saveShowLogStep+10;
		ELSE
			saveShowLogStep:=300;//Done
		END_IF
	ELSE
		saveShowLogStep:=300;//Done
	END_IF
	
60:
	fbShowLogFileWrite(
		sNetId:= , 
		hFile:= hShowLogFile, 
		pWriteBuff:= , 
		cbWriteLen:= , 
		bExecute:= FALSE, 
		tTimeout:= , 
		bBusy=> , 
		bError=> , 
		nErrId=> , 
		cbWrite=> );
		
	saveShowLogStep:=saveShowLogStep+10;
70:	
	fbShowLogFileWrite(
		sNetId:= , 
		hFile:= hShowLogFile, 
		pWriteBuff:= ADR(saveShowLogStrBuff1), 
		cbWriteLen:= TO_UDINT(LEN(saveShowLogStrBuff1)), 
		bExecute:= TRUE, 
		tTimeout:= , 
		bBusy=> , 
		bError=> , 
		nErrId=> , 
		cbWrite=> );
	IF NOT fbShowLogFileWrite.bBusy AND NOT fbShowLogFileWrite.bError THEN
		saveShowLogStep:=50;//返回
		iShowLogTemp:=iShowLogTemp+1;
		fbShowLogFileClose(
			sNetId:= , 
			hFile:= hShowLogFile, 
			bExecute:= FALSE);
	ELSIF fbShowLogFileWrite.bError THEN
		saveShowLogStep:=500;//Error
		fbShowLogFileClose(
			sNetId:= , 
			hFile:= hShowLogFile, 
			bExecute:= FALSE);
	END_IF

300://Done
	fbShowLogFileClose(
		sNetId:= , 
		hFile:= hShowLogFile, 
		bExecute:= TRUE, 
		tTimeout:= , 
		bBusy=> , 
		bError=> , 
		nErrId=> );
	IF NOT fbShowLogFileClose.bBusy THEN
		saveShowLogStep:=saveShowLogStep+1;
	END_IF
301:
	fbShowLogFileClose(
		sNetId:= , 
		hFile:= hShowLogFile, 
		bExecute:= FALSE);
	saveShowLogStep:=0;
	
	bShowLogBusy:=FALSE;
	saveShowLogB:=FALSE;

500://Error
	fbShowLogFileClose(
		sNetId:= , 
		hFile:= hShowLogFile, 
		bExecute:= TRUE, 
		tTimeout:= , 
		bBusy=> , 
		bError=> , 
		nErrId=> );
	IF NOT fbShowLogFileClose.bBusy THEN
		saveShowLogStep:=saveShowLogStep+1;
	END_IF
501:
	fbShowLogFileClose(
		sNetId:= , 
		hFile:= hShowLogFile, 
		bExecute:= FALSE);
	saveShowLogStep:=0;
	
	bShowLogBusy:=FALSE;
	saveShowLogB:=FALSE;
END_CASE
END_METHOD

METHOD PRIVATE showInfo : BOOL
VAR_INPUT
	str				:WSTRING(255):="";
	sTime			:WSTRING(255):="";
END_VAR
VAR
	iTempShowInfo	:DINT;
END_VAR
IF enableShowInfo THEN
	FOR iTempShowInfo:=cNumLength_showInof TO (cNumBegin_showInof+1) BY -1 DO
		HMIData.logStrData[iTempShowInfo]:=HMIData.logStrData[iTempShowInfo-1];
	END_FOR
	HMIData.logStrData[cNumBegin_showInof].sTime:=sTime;
	HMIData.logStrData[cNumBegin_showInof].msg:=str;
END_IF
END_METHOD

ACTION VersionLog:
(*
版本: V1.0.0.0
说明:
	1. 首个版本
	2. 可通过append\append_EX函数添加队列log打印显示
/**************************************************/
版本: V1.0.0.1
说明:
	1. 增加文件自动删除功能
/**************************************************/
*)
END_ACTION

ACTION WPersData:
(* 需要在变量改变之后, PLC断电之前触发bWrtie *)
wrtieR_TRIG(CLK:=bWrtie);

fbGetCurTaskIndex(index=>nTaskNo);
fbWritePersistentData(
	NETID:= , 
	PORT:= 851, 
	START:= wrtieR_TRIG.Q OR TwinCAT_SystemInfoVarList._TaskInfo[nTaskNo].FirstCycle, 
	TMOUT:= , 
	MODE:= , 
	BUSY=> , 
	ERR=> , 
	ERRID=> );

IF wrtieR_TRIG.Q THEN
	bWrtie:=FALSE;
END_IF

(* 以下仅用于带1s UPS的CX51x0 PLC *)
fbUPS(
	sNetID:= , 
	iPLCPort:= 851, 
	iUPSPort:= , 
	tTimeout:= , 
	eUpsMode:= , 
	ePersistentMode:= , 
	tRecoverTime:= , 
	bPowerFailDetect=> , 
	eState=> );
END_ACTION

END_FUNCTION_BLOCK

// ---- POUs/BaseModule/ActionModule/MFCModule/MFCModule.TcPOU
(*
--报错编号0: 无报错
--报错编号1: openend Error
--报错编号2: closeract Error
*)
FUNCTION_BLOCK MFCModule
VAR_IN_OUT
	WarmHMI					:WARMStruct;
	operatorLog				:printLogModule_EX;
END_VAR
VAR_INPUT
	MFCType						:MFCType:=MFCType_Default;// 设置MFC的类型
	MFCHMItif					:MFCStruct;
	set							:BOOL:=FALSE;// 设置触发信号
	setCondition				:BOOL:=TRUE;// 设置触发条件
	clear						:BOOL:=FALSE;// 清零触发信号
	clearCondition				:BOOL:=TRUE;// 清零条件
	reset						:BOOL:=FALSE;// 复位信号
	stop						:BOOL:=FALSE;// 停止信号
	power						:BOOL:=TRUE;// TRUE--保持得电,FALSE--断开得电
	enable						:BOOL:=TRUE;// MFC禁用条件
	//ctrlMode					:ControlMode:=ControlMode.eManualCtrMode;//eManualCtrMode or eAutoCtrMode
	hmiEN						:BOOL:=TRUE;//HMI 启用条件
	
	errorDelayTime				:TIME:=T#2S;// MFC设置参数超时
	
	ACCMaxtime					:TIME:=T#2S;// MFC加速最大时间
	DCCMaxtime					:TIME:=T#2S;// MFC减速最大时间
	
	doneDelayTimeShortset		:TIME:=T#10MS;// MFC设置值到达延时_设置
	doneDelayTimeShortclear		:TIME:=T#10MS;// MFC设置值到达延时_清零
	errorID						:UDINT:=0;// MFC错误报警分配的起始ID
	nameTXT						:STRING(255):='';// MFC名字
	
	AlmAprSw					:BOOL:=FALSE;// 分子泵报警感应器信号,需要链接到实际的IO点
	
	temperatureMax				:REAL;// MFC温度报警设置值
	setFlow						:UDINT;// MFC流量设定
	maxSetValue					:REAL;// MFC流量设定上限
	minSetValue					:REAL;// MFC流量设定下限
	serialSlaveID				:UINT;// MFC ID
	serialError					:BOOL;// MFC通讯错误
	noteWTXT_set				:WSTRING(255):="";// MFC设置动作NoteTXT 中文
	noteWTXT_clear				:WSTRING(255):="";// MFC清零动作NoteTXT 中文
	
	serialExcute				:BOOL;// 通讯数据发送
	connected					:BOOL;
	connectedCount				:UDINT;
	flow					:UDINT;// 设定反馈流量值
	
	actflow					:UDINT;// 实际反馈流量值
	actflowFloat			:REAL;// 实际反馈流量值
END_VAR
VAR_OUTPUT
	note_set				:BOOL;// 设置条件不满足提示
	note_clear				:BOOL;// 清零条件不满足提示
	
	sendBusy				:BOOL;// 串口发送数据繁忙
	
	busy					:BOOL;// MFC动作Busy状态
	setbusy					:BOOL;// MFC设置动作Busy状态
	clearbusy				:BOOL;// MFC清零动作Busy状态
	done					:BOOL;// MFCdone状态
	setdone					:BOOL;// MFC设置完成
	cleardone				:BOOL;// MFC清零完成
	error					:BOOL;//  MFC error状态
	errID					:UDINT;// MFC errID
	errTXT					:STRING(255):='';//  MFC errTXT
	errWTXT					:WSTRING(255):="";//  MFC errTXT 中文
END_VAR
	
VAR	
	setErrorDelayTon		:Ton;
	setDoneDelayTon			:Ton;
	clearErrorDelayTon		:Ton;
	clearDoneDelayTon		:Ton;
	
	setTrigRAlc			    :R_Trig;//上升沿触发
	
	clearTrigRAlc			:R_Trig;//上升沿触发
	
	setTrigR1			:R_Trig;//上升沿触发
	setTrigR1_Aiko		:R_Trig;//上升沿触发
	clearRactTrigR1			:R_Trig;//上升沿触发
	resetTrigR1				:R_Trig;//上升沿触发
	stopTrigR1				:R_Trig;//上升沿触发
	powerTrigR1				:R_Trig;//上升沿触发
	
	setStep					:UINT:=0;
	clearStep				:UINT:=0;
	errorStep				:UINT:=0;
	
	resetRelayTON			:TON;
	resetRelayTONTime		:TIME:=T#2S;
	
	AccFTrig:F_TRIG;//检测加速信号下降延
	DccFTrig:F_TRIG;// 检测减速信号下降延
	noteTON_P:tON;            // 操作提示标志位延时继电器
	noteTON_N:tON;            // 操作提示标志位延时继电器
	noteRTrig_P:R_TRIG;          // 操作提示
	noteRTrig_N:R_TRIG;          // 操作提示
END_VAR

Init_ACT();
Error_ACT();
Set_ACT();
Clear_ACT();
Reset_ACT();
Error_ACT();

(*
触发缩回动作，成功触发返回TRUE，触发失败返回FALSE
*)
METHOD Act_Clear : BOOL
VAR_INPUT
END_VAR
IF enable AND clearCondition THEN// AND NOT busy
	Act_Clear:=clear:=TRUE;
ELSE
	Act_Clear:=FALSE;
END_IF
END_METHOD

(*
触发复位报警动作，成功触发返回TRUE，触发失败返回FALSE
*)
METHOD Act_Reset : BOOL
VAR_INPUT
END_VAR
Act_Reset:=reset:=TRUE;
END_METHOD

(*
触发发送动作，成功触发返回TRUE，触发失败返回FALSE
*)
METHOD Act_SerialSend : BOOL
VAR_INPUT
END_VAR
IF TRUE THEN
	Act_SerialSend:=serialExcute:=TRUE;
ELSE
	Act_SerialSend:=FALSE;
END_IF
END_METHOD

(*
触发伸出动作，成功触发返回TRUE，触发失败返回FALSE
*)
METHOD Act_Set : BOOL
VAR_INPUT
	_setpoint:UDINT;
END_VAR
IF enable AND setCondition THEN// AND NOT busy
	setFlow:=_setpoint;
	Act_Set:=set:=TRUE;
ELSE
	Act_Set:=FALSE;
END_IF
END_METHOD

(*
触发停止输出动作，成功触发返回TRUE，触发失败返回FALSE
*)
METHOD Act_Stop : BOOL
VAR_INPUT
END_VAR
Act_Stop:=stop:=TRUE;
END_METHOD

ACTION Clear_ACT:
//MFC--clear 触发
IF clear AND NOT clearCondition THEN
	note_set:=FALSE;
	note_clear:=TRUE;
END_IF
IF clear AND enable AND NOT error AND clearCondition AND NOT clearbusy AND NOT gMFCStopLoopRead THEN// AND NOT busy
	note_set:=FALSE;
	note_clear:=FALSE;
	busy:=TRUE;
	clearbusy:=TRUE;
	setbusy:=FALSE;
	set:=FALSE;
	setdone:=FALSE;
	cleardone:=FALSE;
	setStep:=0;
	clearStep:=10;
	gMFCStopLoopRead:=TRUE;
	operatorLog.append(CONCAT(nameTXT,' Clear'));
	//errorStep:=0;
END_IF
clear:=FALSE;

CASE clearStep OF
0:
	//ready
	
10:
	IF FuncModule_RS485_MFC.loopReadStep<10 OR FuncModule_RS485_MFC.loopReadStep>270 THEN
		clearErrorDelayTon(IN:=FALSE);
		clearDoneDelayTon(IN:=FALSE);
		clearStep:=20;
		setFlow:=0;
		FuncModule_RS485_MFC.Interface_Set(serialSlaveID,setFlow);
	END_IF
	
20:
	clearErrorDelayTon(IN:=(NOT FuncModule_RS485_MFC.setDone ),PT:=errorDelayTime);
	IF clearErrorDelayTon.Q THEN
		//done:=FALSE;
		setdone:=FALSE;
		cleardone:=FALSE;
		errorStep:=2;
		clearStep:=60;
		clearbusy:=FALSE;
		setbusy:=FALSE;
		RETURN;
	END_IF
	clearDoneDelayTon(IN:=FuncModule_RS485_MFC.setDone,PT:=doneDelayTimeShortclear);
	IF clearDoneDelayTon.Q THEN
		clearErrorDelayTon(IN:=FALSE);
		clearDoneDelayTon(IN:=FALSE);
		setFlow:=0;
		// send Set point
		clearStep:=30;
	END_IF
30:
	IF NOT error THEN
		busy:=FALSE;
		clearbusy:=FALSE;
		setbusy:=FALSE;
		//done:=TRUE;
		setdone:=FALSE;
		cleardone:=TRUE;
		errorStep:=0;
		clearStep:=50;
		gMFCStopLoopRead:=FALSE;
	ELSE
		busy:=FALSE;
		clearbusy:=FALSE;
		setbusy:=FALSE;
		//done:=TRUE;
		setdone:=FALSE;
		cleardone:=FALSE;
		errorStep:=3;
		clearStep:=60;
		gMFCStopLoopRead:=FALSE;
	END_IF
END_CASE
END_ACTION

ACTION Error_ACT:
CASE errorStep OF
	0:
		error:=FALSE;
		errID:=0;
		errTXT:='';
 (*
	1:
		error:=TRUE;
		errID:=errorID+errorStep;
		errTXT:=CONCAT(STR1:=nameTXT,STR2:=' Extend Error!');
		errWTXT:=WCONCAT(STR1:=TO_WSTRING(nameTXT),STR2:=" 伸出(打开)错误");
	2:
		error:=TRUE;
		errID:=errorID+errorStep;
		errTXT:=CONCAT(STR1:=nameTXT,STR2:=' Retract Error!');
		errWTXT:=WCONCAT(STR1:=TO_WSTRING(nameTXT),STR2:=" 缩回(关闭)错误");
		*)
	1..5:
		error:=TRUE;
		errID:=getErrID(errorStep);
		errTXT:=getErrTXT(errorStep);
		errWTXT:=getErrWTXT(errorStep);
END_CASE
END_ACTION

METHOD Get_Done_Clear : BOOL
VAR_INPUT
END_VAR
Get_Done_Clear:=cleardone;
END_METHOD

METHOD Get_Done_Set : BOOL
VAR_INPUT
END_VAR
Get_Done_Set:=setdone;
END_METHOD

METHOD getErrID : UDINT
VAR_INPUT
	errID					:UDINT;//取值范围1~2
END_VAR
VAR
	nErrID					:UDINT;
END_VAR
nErrID:=errorID+errID;

getErrID:=nErrID;
END_METHOD

METHOD getErrTXT : STRING(255)
VAR_INPUT
	errID					:UDINT;//取值范围1~2
END_VAR
VAR
	sErrTXT					:STRING(255);
END_VAR

CASE errID OF
	1:
		sErrTXT:=CONCAT(STR1:=nameTXT,STR2:=' Set Error!');
	2:
		sErrTXT:=CONCAT(STR1:=nameTXT,STR2:=' Clear Error!');
	3:
		sErrTXT:=CONCAT(STR1:=nameTXT,STR2:=' NormalRun Error!');
	4:
		sErrTXT:=CONCAT(STR1:=nameTXT,STR2:=' SetValue Error!');
	5:
		sErrTXT:=CONCAT(STR1:=nameTXT,STR2:=' IO Fault!');
ELSE
	sErrTXT:=CONCAT(STR1:=nameTXT,STR2:='');
END_CASE
getErrTXT:=sErrTXT;
END_METHOD

METHOD getErrWTXT : WSTRING(255)
VAR_INPUT
	errID					:UDINT;//取值范围1~16
END_VAR
VAR
	sErrTXT					:WSTRING(255);
END_VAR

CASE errID OF
	1:
		sErrTXT:=WCONCAT(STR1:=TO_WSTRING(nameTXT),STR2:="  设置 错误");
	2:
		sErrTXT:=WCONCAT(STR1:=TO_WSTRING(nameTXT),STR2:="  清零 错误");
	3:
		sErrTXT:=WCONCAT(STR1:=TO_WSTRING(nameTXT),STR2:="  正常运行出现异常情况");
	4:
		sErrTXT:=WCONCAT(STR1:=TO_WSTRING(nameTXT),STR2:="  参数设置出错");
	5:
		sErrTXT:=WCONCAT(STR1:=TO_WSTRING(nameTXT),STR2:="  IO报错");
ELSE
	sErrTXT:=WCONCAT(STR1:=TO_WSTRING(nameTXT),STR2:="");
END_CASE
getErrWTXT:=sErrTXT;
END_METHOD

ACTION Init_ACT:
done:=(cleardone OR setdone);
IF AlmAprSw THEN
	errorStep:=5;
END_IF
error:=error OR serialError OR AlmAprSw;
manualCtrl_ACT();
IF (error OR AlmAprSw OR serialError) AND flow>0.1 THEN
	stop:=TRUE;
	busy:=FALSE;
END_IF

noteTON_P(IN:=note_set,PT:=T#0.1S);
noteRTrig_P(CLK:=noteTON_P.Q);
IF noteRTrig_P.Q THEN
	//gLog_Note.append_EX(noteWTXT_Open);
	;
END_IF
noteTON_N(IN:=note_clear,PT:=T#0.1S);
noteRTrig_N(CLK:=noteTON_N.Q);
IF noteRTrig_N.Q THEN
	//gLog_Note.append_EX(noteWTXT_close);
	;
END_IF
END_ACTION

ACTION ManualCtrl_ACT:
////HMI手动控制
////IF ctrlMode=eManualCtrMode THEN
IF hmiEN THEN
	setTrigR1(CLK:=MFCHMItif.set);
	IF setTrigR1.Q THEN
		MFCHMItif.set:=FALSE;
		WarmHMI.showText:='';
		WarmHMI.showFlag:=TRUE;
		WarmHMI.showText:=CONCAT(WarmHMI.showText,'Are you sure you want ');
		WarmHMI.showText:=CONCAT(WarmHMI.showText,nameTXT);
		WarmHMI.showText:=CONCAT(WarmHMI.showText,' to Set it?');
	END_IF
	IF WarmHMI.bOK AND NOT WarmHMI.showFlag AND FIND(WarmHMI.showText,nameTXT)>0 AND FIND(WarmHMI.showText,'Set')>0 THEN
		set:=TRUE;
		WarmHMI.bOK:=FALSE;
		WarmHMI.showText:='';
	END_IF
	IF WarmHMI.bNO AND NOT WarmHMI.showFlag AND FIND(WarmHMI.showText,nameTXT)>0 AND FIND(WarmHMI.showText,'Set')>0 THEN
		WarmHMI.bNO:=FALSE;
		MFCHMItif.set:=FALSE;
		WarmHMI.showText:='';
	END_IF
	clearTrigRAlc(CLK:=MFCHMItif.clear);
	IF clearTrigRAlc.Q THEN
		MFCHMItif.clear:=FALSE;
		WarmHMI.showText:='';
		WarmHMI.showFlag:=TRUE;
		WarmHMI.showText:=CONCAT(WarmHMI.showText,'Are you sure you want to Clear the ');
		WarmHMI.showText:=CONCAT(WarmHMI.showText,nameTXT);
		WarmHMI.showText:=CONCAT(WarmHMI.showText,' `Par?');
	END_IF
	IF WarmHMI.bOK AND NOT WarmHMI.showFlag AND FIND(WarmHMI.showText,nameTXT)>0 AND FIND(WarmHMI.showText,'Clear')>0 THEN
		clear:=TRUE;
		WarmHMI.bOK:=FALSE;
		WarmHMI.showText:='';
	END_IF
	IF WarmHMI.bNO AND NOT WarmHMI.showFlag AND FIND(WarmHMI.showText,nameTXT)>0 AND FIND(WarmHMI.showText,'Clear')>0 THEN
		WarmHMI.bNO:=FALSE;
		MFCHMItif.clear:=FALSE;
		WarmHMI.showText:='';
	END_IF
END_IF
END_ACTION

ACTION Reset_ACT:
IF reset THEN
	note_set:=FALSE;
	note_clear:=FALSE;
	setStep:=0;
	clearStep:=0;
	errorStep:=0;
	reset:=FALSE;
END_IF
//resetRelayTON(IN:=resetRelay , PT:=resetRelayTONTime);
//IF resetRelayTON.Q THEN
//	openStep:=0;
//	closeStep:=0;
//	errorStep:=0;
//	busy:=FALSE;
//	resetRelay:=FALSE;
//END_IF

//IF stop THEN
//	note_open:=FALSE;
//	note_close:=FALSE;
//	stop:=FALSE;
//	openRelay:=FALSE;
//	closeRelay:=FALSE;
//	//无自锁检测说法，直接停
//	openStep:=0;
//	closeStep:=0;
//END_IF
END_ACTION

ACTION Serial_Act:
//(*
// *功能块的作用，把 TxBuffer 缓存区的数据经过 Process Data 的 ComOut 发送出去，
// *而把 ComIn 中的数据接收到 RxBuffer。引用这个功能块的程序执行周期越短，
// *数据交换的效率就越高，所以这段程序应该放在快速任务中作为 Backgroud 代码无条件执行。
//*)
//COMportControl(
//	Mode:= SERIALLINEMODE_KL6_22B_STANDARD, 
//	pComIn:= ADR(COMin), 
//	pComOut:= ADR(COMout), 
//	SizeComIn:= SIZEOF(COMin), 
//	Error=> , 
//	ErrorID=> , 
//	TxBuffer:= TxBuffer_TMP, 
//	RxBuffer:= RxBuffer_TMP );
//IF receive1.Error <> COMERROR_NOERROR THEN
//	serialRecError:=TRUE;
//END_IF
//receive1(
//	pPrefix:= , 
//	LenPrefix:= , 
//	pSuffix:= , 
//	LenSuffix:= , 
//	pReceiveData:= ADR(arr_RcvData), 
//	SizeReceiveData:= 100, 
//	Timeout:= T#100MS, //临时设置成10S调试用
//	Reset:= , 
//	DataReceived=> , 
//	busy=> , 
//	Error=> , 
//	RxTimeout=> , 
//	LenReceiveData=> , 
//	RXbuffer:= RxBuffer_TMP);
////testReal:=BYTE_TO_REAL(arr_RcvData_Temp);
//CASE serialStep OF
//	0:
//	IF enableSerial AND serialExcute THEN
//		serialExcute:=FALSE;
//		IF NOT serialBusy THEN
//			serialStep:=10;
//			serialBusy:=TRUE;
//			serialDone:=FALSE;
//			serialError:=FALSE;
//			serialTimeOut:=FALSE;
//			serialRecError:=FALSE;
//			receive1(//复位
//				pPrefix:= , 
//				LenPrefix:= , 
//				pSuffix:= , 
//				LenSuffix:= , 
//				pReceiveData:= , 
//				SizeReceiveData:=, 
//				Timeout:= T#300MS, 
//				Reset:= , 
//				DataReceived=> , 
//				busy=> , 
//				Error=> , 
//				RxTimeout=> , 
//				LenReceiveData=> , 
//				RXbuffer:= RxBuffer_TMP);
//		END_IF
//	END_IF
//	Timer1(IN:= FALSE);
//	;
//	10:
//		//第二和第三位代表ID号
//		arr_SendData[1]	:=16#40;
//		IF serialSlaveID>9 THEN
//			arr_SendData[2]	:=F_ToASC(str:='0');
//			arr_SendData[3]	:=F_ToASC(str:=(UINT_TO_STRING(serialSlaveID)));
//		ELSE
//			arr_SendData[2]	:=F_ToASC(str:=(UINT_TO_STRING(serialSlaveID/10)));
//			arr_SendData[3]	:=F_ToASC(str:=(UINT_TO_STRING(serialSlaveID MOD 10)));
//		END_IF
//		arr_SendData[4]:=16#02;
//		arr_SendData[5]:=16#30;
//		arr_SendData[6]:=16#30;
//		arr_SendData[7]:=16#31;
//		arr_SendData[8]:=16#3F;
//		arr_SendData[9]:=16#5B;
//		arr_SendData[10]:=16#03;
//		arr_SendData[11]:=16#AB;
//		serialStep:=100;
//	100:
//		send1(
//			pSendData:= ADR(arr_SendData), 
//			Length:= nSendByteLength, 
//			Busy=> , 
//			Error=> , 
//			TXbuffer:= TxBuffer_TMP);
//		serialStep:=serialStep+20;
//	110:
//		Timer1(IN:= NOT timer1.q, PT:=T#00MS);
//		IF Timer1.Q THEN
//			serialStep:=serialStep+10;
//			Timer1(IN:= FALSE);
//		END_IF
//	120:
//		Timer1(IN:= NOT timer1.q, PT:=T#3000MS);
//		IF Timer1.Q THEN
//			serialStep:=6000;
//			Timer1(IN:= FALSE);
//			serialTimeOut:=TRUE;
//			RETURN;
//		END_IF
//		IF receive1.DataReceived THEN
//			Timer1(IN:= FALSE);
//			serialTimeOut:=FALSE;
//			serialStep:=200;
//		END_IF
//		IF receive1.Error <> COMERROR_NOERROR THEN
//			serialRecError:=TRUE;
//		END_IF
//	200://数据处理
//		arr_RcvData_Temp:=arr_RcvData;
//		arr_RcvData:=arr_RcvData_Clear;
//		serialStep:=serialStep+10;
//	210:
//		//第二和第三位代表ID号;看情况决定是否需要判断节点反馈的节点号
//		IF arr_RcvData_Temp[12]=arr_SendData[9] AND arr_RcvData_Temp[2]=arr_SendData[2] AND arr_RcvData_Temp[3]=arr_SendData[3] THEN
//			serialStep:=serialStep+10;
//			serialRecError:=FALSE;
//		ELSE//数据接线错误
//			serialStep:=6000;
//			serialRecError:=TRUE;
//		END_IF
//	220:
//		//数据转换
//		serialStep:=300;
//	;
//	300:
//		strTemp:='';
//		strTemp:=CONCAT(strTemp,F_TOCHR(arr_RcvData_Temp[47]));
//		strTemp:=CONCAT(strTemp,F_TOCHR(arr_RcvData_Temp[48]));
//		strTemp:=CONCAT(strTemp,F_TOCHR(arr_RcvData_Temp[49]));
//		strTemp:=CONCAT(strTemp,F_TOCHR(arr_RcvData_Temp[50]));
//		temperature:=STRING_TO_UINT(strTemp)*1.0;
//		strTemp:='';
//		strTemp:=CONCAT(strTemp,F_TOCHR(arr_RcvData_Temp[53]));
//		strTemp:=CONCAT(strTemp,F_TOCHR(arr_RcvData_Temp[54]));
//		currentTemp:=STRING_TO_INT(strTemp);
//		current:=INT_TO_REAL(currentTemp)/10.0;// 1位小数
//		strTemp:='';
//		strTemp:=CONCAT(strTemp,F_TOCHR(arr_RcvData_Temp[61]));
//		strTemp:=CONCAT(strTemp,F_TOCHR(arr_RcvData_Temp[62]));
//		strTemp:=CONCAT(strTemp,F_TOCHR(arr_RcvData_Temp[63]));
//		strTemp:=CONCAT(strTemp,F_TOCHR(arr_RcvData_Temp[64]));
//		speed:=STRING_TO_UINT(strTemp)*1.0;
//		serialStep:=5000;
//	;
//	5000://done
//		serialBusy:=FALSE;
//		serialDone:=TRUE;
//		serialError:=FALSE;
//		serialStep:=0;
//	;
//	6000://error
//		serialBusy:=FALSE;
//		serialDone:=FALSE;
//		serialError:=TRUE;
//		serialStep:=0;
//	;
	
//END_CASE
////arr_Temp[1]:=arr_RcvData_Temp[48];
////arr_Temp[2]:=arr_RcvData_Temp[47];
////MEMMOVE(ADR(temperatureTemp),ADR(arr_Temp[1]),2);// 2个字节
////temperature:=DINT_TO_REAL(temperatureTemp);
////MEMMOVE(ADR(currentTemp),ADR(arr_RcvData_Temp[53]),1);// 1个字节
////current:=INT_TO_REAL(currentTemp)/1.0;// 1位小数
////arr_Temp1[1]:=arr_RcvData_Temp[62];
////arr_Temp1[2]:=arr_RcvData_Temp[61];
////MEMMOVE(ADR(speedTemp),ADR(arr_Temp1[1]),2);// 2个字节
////speed:=DINT_TO_REAL(speedTemp);
////speed:=speed*60.0;
////IF enableSerial THEN//启用
////	;
////	 //字符串方式
////	 (*//3000ms发送一次
////	Timer1(IN:= NOT timer1.q, PT:=T#3000MS , Q=> , ET=> );
////	IF timer1.Q THEN
////		SEND1(
////			SendString:=_sendString ,
////			TXbuffer:=TxBuffer_TMP ,
////			Busy=> ,
////			Error=> );
////	END_IF
	 
////	//接收
////	Receive1(
////		Timeout:= t#100ms,
////		ReceivedString:=_receive1string ,
////		RXbuffer:=RxBuffer_TMP , );
	 
////	//保存上一个周期接收的字符
////	IF Receive1.Busy THEN
////		_recvLast:=_receive1string;
////	END_IF*)
////END_IF
END_ACTION

ACTION Set_ACT:
//MFC--set 触发
IF set AND NOT setCondition THEN
	note_clear:=FALSE;
	note_set:=TRUE;
END_IF
IF set AND enable AND NOT error AND setCondition AND NOT setbusy AND NOT gMFCStopLoopRead THEN// AND NOT busy
	note_set:=FALSE;
	note_clear:=FALSE;
	busy:=TRUE;
	setbusy:=TRUE;
	clearbusy:=FALSE;
	set:=FALSE;
	setdone:=FALSE;
	cleardone:=FALSE;
	setStep:=10;
	clearStep:=0;
	gMFCStopLoopRead:=TRUE;
	operatorLog.append(CONCAT(CONCAT(nameTXT,' Set '),UDINT_TO_STRING(setFlow)));
	//errorStep:=0;
END_IF
set:=FALSE;

CASE setStep OF
0:
	//ready

10:
 	IF FuncModule_RS485_MFC.loopReadStep<10 OR FuncModule_RS485_MFC.loopReadStep>270 THEN
		setErrorDelayTon(IN:=FALSE);
		setDoneDelayTon(IN:=FALSE);
		IF (UDINT_TO_REAL(setFlow)<=maxSetValue AND UDINT_TO_REAL(setFlow)>=minSetValue) THEN
			setStep:=20;
			FuncModule_RS485_MFC.Interface_Set(serialSlaveID,setFlow);
		ELSE
			setdone:=FALSE;
			cleardone:=FALSE;
			setStep:=60;
			gMFCStopLoopRead:=FALSE;
			errorStep:=4;
			setFlow:=flow;
			clearbusy:=FALSE;
			setbusy:=FALSE;
			setDoneDelayTon(IN:=FALSE);
			setErrorDelayTon(IN:=FALSE);
		END_IF
	END_IF
20:
	setErrorDelayTon(IN:=(NOT FuncModule_RS485_MFC.setDone ),PT:=errorDelayTime);
	IF setErrorDelayTon.Q THEN
		//done:=FALSE;
		setdone:=FALSE;
		cleardone:=FALSE;
		errorStep:=1;
		setStep:=60;
		gMFCStopLoopRead:=FALSE;
		clearbusy:=FALSE;
		setbusy:=FALSE;
		RETURN;
	END_IF
	setDoneDelayTon(IN:=FuncModule_RS485_MFC.setDone,PT:=doneDelayTimeShortset);
	IF setDoneDelayTon.Q THEN
		setErrorDelayTon(IN:=FALSE);
		setDoneDelayTon(IN:=FALSE);
		setStep:=30;
	END_IF
30:
	IF NOT error THEN
		busy:=FALSE;
		clearbusy:=FALSE;
		setbusy:=FALSE;
		//done:=TRUE;
		cleardone:=FALSE;
		setdone:=TRUE;
		errorStep:=0;
		setStep:=50;
		gMFCStopLoopRead:=FALSE;
	ELSE
		busy:=FALSE;
		clearbusy:=FALSE;
		setbusy:=FALSE;
		//done:=TRUE;
		setdone:=FALSE;
		cleardone:=FALSE;
		errorStep:=3;
		setFlow:=flow;
		setStep:=60;
		gMFCStopLoopRead:=FALSE;
	END_IF

END_CASE
END_ACTION

ACTION VersionLog:
(*
版本: V1.0.0.0
说明:
	1. 首个版本
	2. 含普通分子泵\泵组类型的控制
	3. 可配置是否有到位信号, 以及到位稳定时间
*)
END_ACTION

END_FUNCTION_BLOCK

// ---- POUs/BaseModule/Communication/FuncModule_RS485_MFC.TcPOU
PROGRAM FuncModule_RS485_MFC
VAR_INPUT
	serialExcute				:BOOL;// RS485开始一次参数读取
	setExcute					:BOOL;// RS485
	readExcute					:BOOL;// RS485
	serialSlaveID				:UDINT:=1;// 从站节点号
	sendLenght					:UINT:=14;// 发送字节长度
	sendbyte					:ARRAY[1..20]			OF		BYTE;(*READ*)//发送数据
	timeout						:TIME:=T#100MS;// 超时时间
	setPoint					:UDINT;
	loopReadStep				:INT;
	loopReadExcute				:BOOL;
	loopReadIntervalTime		:UDINT:=0;
END_VAR
VAR_OUTPUT
	serialBusy						:BOOL;
	setPresetBusy					:BOOL;
	serialDone						:BOOL;
	serialError						:BOOL;
	serialConnected					:BOOL;
	setBusy							:BOOL;// 设置参数时繁忙
	setError						:BOOL;
	setDone							:BOOL;
	readBusy						:BOOL;// 读取参数时繁忙
	readError						:BOOL;
	readDone						:BOOL;
	readID							:BOOL;
END_VAR
VAR
	
	prefix						:STRING:='';// 字符串头
	suffix						:STRING:= '';// 字符串尾
	readsetStarIndex				:INT;
	readsetPointStarIndex				:INT;
	readsetPointEndIndex				:INT;
	readsetPointStr				:STRING;
	readPointStr				:STRING;
	readIDStr					:STRING;
	readPointReal				:LREAL;
	readPointInt				:UDINT;
	
	readIDInt							:UDINT;
	//Byte方式
	send1:							SendData;
	receive1:						ReceiveString;
	Timer1:							TON;
	TimerSetPreset:							TON;
	TimerReadPreset:							TON;
	t1:								TON;
	arr_SendData:					ARRAY[1..20]			OF		BYTE;(*READ*)//发送数据
	arr_SendDataTemp				:ARRAY[1..20]			OF		BYTE;(*READ*)//发送数据
	arr_RcvDataString:				STRING;// 接收数据
	arr_RcvDataStringTemp:				STRING;// 接收数据
	arr_RcvDataStringClear:			STRING;// 清除接收数据
	RcvDataFlag:			BOOL;// 接收数据标志位
	serialStep						:UINT;				//处理步数
	setPresetStep					:UINT;				//处理步数
	readflowStep					:UINT;				//处理步数
	serialTimeOut:BOOL;//接收数据超时
	serialRecError:BOOL;//接收数据错误
	reciveFtrig:F_TRIG;
	recTon:TON;
	againSendS3:TON;
	hexChars:ARRAY [0..15] OF STRING[1]:=['0','1','2','3','4','5','6','7','8','9','A','B','C','D','E','F'];
END_VAR

(*
 *功能块的作用，把 TxBuffer 缓存区的数据经过 Process Data 的 ComOut 发送出去，
 *而把 ComIn 中的数据接收到 RxBuffer。引用这个功能块的程序执行周期越短，
 *数据交换的效率就越高，所以这段程序应该放在快速任务中作为 Backgroud 代码无条件执行。
*)
IF receive1.Error <> COMERROR_NOERROR THEN
	serialRecError:=TRUE;
END_IF
receive1(
	Prefix:= prefix, 
	Suffix:= suffix, 
	Timeout:=timeout , 
	Reset:= , 
	StringReceived=> , 
	Busy=> , 
	Error=> , 
	RxTimeout=> , 
	ReceivedString:= arr_RcvDataStringTemp, 
	RXbuffer:=gRxBuffer_MFC );

//testReal:=BYTE_TO_REAL(arr_RcvData_Temp);
//数据接收处理
recTon(IN:=RcvDataFlag, PT:=T#10MS);
IF recTon.Q THEN
	RcvDataFlag:=FALSE;
END_IF
reciveFtrig(CLK:=receive1.busy);
IF reciveFtrig.Q THEN
	arr_RcvDataString:=arr_RcvDataStringTemp;
	arr_RcvDataStringTemp:=arr_RcvDataStringClear;
	RcvDataFlag:=TRUE;
	serialConnected:=TRUE;
END_IF
againSendS3(IN:=NOT RcvDataFlag,PT:=T#5S);
IF againSendS3.Q THEN
	serialConnected:=FALSE;
	againSendS3(IN:=FALSE);
END_IF
ACT_Send();
ACT_Set();
ACT_Read();
ACT_MFCRead();

ACTION ACT_MFCRead:
IF NOT setBusy AND NOT serialBusy AND NOT readBusy AND NOT gMFCStopLoopRead THEN
	loopReadExcute:=TRUE;
END_IF
CASE loopReadStep OF
	0:
		IF loopReadExcute THEN
			loopReadExcute:=FALSE;
			loopReadStep:=10;
		END_IF
		t1(IN:=FALSE);
	10:
		IF NOT gMFCStopLoopRead THEN
			Interface_Read(1);
			t1(IN:=FALSE);
			loopReadStep:=loopReadStep+10;
		ELSE
			loopReadStep:=5000;
		END_IF
	20:
		IF readDone THEN
			loopReadStep:=loopReadStep+10;
			gICP.MFC1.connected:=TRUE;
			gICP.MFC1.connectedCount:=0;
			gICP.MFC1.actflowFloat:=ReadLLimit(LREAL_TO_REAL(readPointReal));
			gICP.MFC1.actflow:=REAL_TO_UDINT(gICP.MFC1.actflowFloat);
			t1(IN:=FALSE);
			RETURN;
		END_IF
		t1(IN:=TRUE,PT:=T#200MS);
		IF t1.Q THEN
			gICP.MFC1.connectedCount:=gICP.MFC1.connectedCount+1;
			IF gICP.MFC1.connectedCount>10 THEN
				gICP.MFC1.connectedCount:=0;
				gICP.MFC1.connected:=FALSE;
				loopReadStep:=loopReadStep+10;
			ELSE
				loopReadStep:=loopReadStep+10;
			END_IF
			t1(IN:=FALSE);
		END_IF
	30:
		t1(IN:=TRUE,PT:=UDINT_TO_TIME(loopReadIntervalTime));
		IF t1.Q THEN
			loopReadStep:=loopReadStep+10;
			t1(IN:=FALSE);
		END_IF
	40:
		IF NOT gMFCStopLoopRead THEN
			Interface_Read(2);
			t1(IN:=FALSE);
			loopReadStep:=loopReadStep+10;
		ELSE
			loopReadStep:=5000;
		END_IF
	50:
		IF readDone THEN
			loopReadStep:=loopReadStep+10;
			gICP.MFC2.connected:=TRUE;
			gICP.MFC2.connectedCount:=0;
			gICP.MFC2.actflowFloat:=ReadLLimit(LREAL_TO_REAL(readPointReal));
			gICP.MFC2.actflow:=REAL_TO_UDINT(gICP.MFC2.actflowFloat);
			t1(IN:=FALSE);
			RETURN;
		END_IF
		t1(IN:=TRUE,PT:=T#200MS);
		IF t1.Q THEN
			gICP.MFC2.connectedCount:=gICP.MFC2.connectedCount+1;
			IF gICP.MFC2.connectedCount>10 THEN
				gICP.MFC2.connectedCount:=0;
				gICP.MFC2.connected:=FALSE;
				loopReadStep:=loopReadStep+10;
			ELSE
				loopReadStep:=loopReadStep+10;
			END_IF
			t1(IN:=FALSE);
		END_IF
	60:
		t1(IN:=TRUE,PT:=UDINT_TO_TIME(loopReadIntervalTime));
		IF t1.Q THEN
			loopReadStep:=loopReadStep+10;
			t1(IN:=FALSE);
		END_IF
	70:
		IF NOT gMFCStopLoopRead THEN
			Interface_Read(3);
			t1(IN:=FALSE);
			loopReadStep:=loopReadStep+10;
		ELSE
			loopReadStep:=5000;
		END_IF
	80:
		IF readDone THEN
			loopReadStep:=loopReadStep+10;
			gICP.MFC3.connected:=TRUE;
			gICP.MFC3.connectedCount:=0;
			gICP.MFC3.actflowFloat:=ReadLLimit(LREAL_TO_REAL(readPointReal));
			gICP.MFC3.actflow:=REAL_TO_UDINT(gICP.MFC3.actflowFloat);
			t1(IN:=FALSE);
			RETURN;
		END_IF
		t1(IN:=TRUE,PT:=T#200MS);
		IF t1.Q THEN
			gICP.MFC3.connectedCount:=gICP.MFC3.connectedCount+1;
			IF gICP.MFC3.connectedCount>10 THEN
				gICP.MFC3.connectedCount:=0;
				gICP.MFC3.connected:=FALSE;
				loopReadStep:=loopReadStep+10;
			ELSE
				loopReadStep:=loopReadStep+10;
			END_IF
			t1(IN:=FALSE);
		END_IF
	90:
		t1(IN:=TRUE,PT:=UDINT_TO_TIME(loopReadIntervalTime));
		IF t1.Q THEN
			loopReadStep:=loopReadStep+10;
			t1(IN:=FALSE);
		END_IF
	100:
		IF NOT gMFCStopLoopRead THEN
			Interface_Read(4);
			t1(IN:=FALSE);
			loopReadStep:=loopReadStep+10;
		ELSE
			loopReadStep:=5000;
		END_IF
	110:
		IF readDone THEN
			loopReadStep:=loopReadStep+10;
			gICP.MFC4.connected:=TRUE;
			gICP.MFC4.connectedCount:=0;
			t1(IN:=FALSE);
			gICP.MFC4.actflowFloat:=ReadLLimit(LREAL_TO_REAL(readPointReal));
			gICP.MFC4.actflow:=REAL_TO_UDINT(gICP.MFC4.actflowFloat);
			RETURN;
		END_IF
		t1(IN:=TRUE,PT:=T#200MS);
		IF t1.Q THEN
			gICP.MFC4.connectedCount:=gICP.MFC4.connectedCount+1;
			IF gICP.MFC4.connectedCount>10 THEN
				gICP.MFC4.connectedCount:=0;
				gICP.MFC4.connected:=FALSE;
				loopReadStep:=loopReadStep+10;
			ELSE
				loopReadStep:=loopReadStep+10;
			END_IF
			t1(IN:=FALSE);
		END_IF
	120:
		t1(IN:=TRUE,PT:=UDINT_TO_TIME(loopReadIntervalTime));
		IF t1.Q THEN
			loopReadStep:=loopReadStep+10;
			t1(IN:=FALSE);
		END_IF
	130:
		IF NOT gMFCStopLoopRead THEN
			Interface_Read(5);
			t1(IN:=FALSE);
			loopReadStep:=loopReadStep+10;
		ELSE
			loopReadStep:=5000;
		END_IF
	140:
		IF readDone THEN
			loopReadStep:=loopReadStep+10;
			gICP.MFC5.connected:=TRUE;
			gICP.MFC5.connectedCount:=0;
			t1(IN:=FALSE);
			gICP.MFC5.actflowFloat:=ReadLLimit(LREAL_TO_REAL(readPointReal));
			gICP.MFC5.actflow:=REAL_TO_UDINT(gICP.MFC5.actflowFloat);
			RETURN;
		END_IF
		t1(IN:=TRUE,PT:=T#200MS);
		IF t1.Q THEN
			gICP.MFC5.connectedCount:=gICP.MFC5.connectedCount+1;
			IF gICP.MFC5.connectedCount>10 THEN
				gICP.MFC5.connectedCount:=0;
				gICP.MFC5.connected:=FALSE;
				loopReadStep:=loopReadStep+10;
			ELSE
				loopReadStep:=loopReadStep+10;
			END_IF
			t1(IN:=FALSE);
		END_IF
	150:
		t1(IN:=TRUE,PT:=UDINT_TO_TIME(loopReadIntervalTime));
		IF t1.Q THEN
			loopReadStep:=loopReadStep+10;
			t1(IN:=FALSE);
		END_IF
	160:
		IF NOT gMFCStopLoopRead THEN
			Interface_Read(6);
			t1(IN:=FALSE);
			loopReadStep:=loopReadStep+10;
		ELSE
			loopReadStep:=5000;
		END_IF
	170:
		IF readDone THEN
			loopReadStep:=loopReadStep+10;
			gICP.MFC6.connected:=TRUE;
			gICP.MFC6.connectedCount:=0;
			t1(IN:=FALSE);
			gICP.MFC6.actflowFloat:=ReadLLimit(LREAL_TO_REAL(readPointReal));
			gICP.MFC6.actflow:=REAL_TO_UDINT(gICP.MFC6.actflowFloat);
			RETURN;
		END_IF
		t1(IN:=TRUE,PT:=T#200MS);
		IF t1.Q THEN
			gICP.MFC6.connectedCount:=gICP.MFC6.connectedCount+1;
			IF gICP.MFC6.connectedCount>10 THEN
				gICP.MFC6.connectedCount:=0;
				gICP.MFC6.connected:=FALSE;
				loopReadStep:=loopReadStep+10;
			ELSE
				loopReadStep:=loopReadStep+10;
			END_IF
			t1(IN:=FALSE);
		END_IF
	180:
		t1(IN:=TRUE,PT:=UDINT_TO_TIME(loopReadIntervalTime));
		IF t1.Q THEN
			loopReadStep:=loopReadStep+10;
			t1(IN:=FALSE);
		END_IF
	190:
		IF NOT gMFCStopLoopRead THEN
			Interface_Read(7);
			t1(IN:=FALSE);
			loopReadStep:=loopReadStep+10;
		ELSE
			loopReadStep:=5000;
		END_IF
	200:
		IF readDone THEN
			loopReadStep:=loopReadStep+10;
			gICP.MFC7.connected:=TRUE;
			gICP.MFC7.connectedCount:=0;
			t1(IN:=FALSE);
			gICP.MFC7.actflowFloat:=ReadLLimit(LREAL_TO_REAL(readPointReal));
			gICP.MFC7.actflow:=REAL_TO_UDINT(gICP.MFC7.actflowFloat);
			RETURN;
		END_IF
		t1(IN:=TRUE,PT:=T#200MS);
		IF t1.Q THEN
			gICP.MFC7.connectedCount:=gICP.MFC7.connectedCount+1;
			IF gICP.MFC7.connectedCount>10 THEN
				gICP.MFC7.connectedCount:=0;
				gICP.MFC7.connected:=FALSE;
				loopReadStep:=loopReadStep+10;
			ELSE
				loopReadStep:=loopReadStep+10;
			END_IF
			t1(IN:=FALSE);
		END_IF
	210:
		t1(IN:=TRUE,PT:=UDINT_TO_TIME(loopReadIntervalTime));
		IF t1.Q THEN
			loopReadStep:=loopReadStep+10;
			t1(IN:=FALSE);
		END_IF
	220:
		IF NOT gMFCStopLoopRead THEN
			Interface_Read(8);
			t1(IN:=FALSE);
			loopReadStep:=loopReadStep+10;
		ELSE
			loopReadStep:=5000;
		END_IF
	230:
		IF readDone THEN
			loopReadStep:=loopReadStep+10;
			gICP.MFC8.connected:=TRUE;
			gICP.MFC8.connectedCount:=0;
			t1(IN:=FALSE);
			gICP.MFC8.actflowFloat:=ReadLLimit(LREAL_TO_REAL(readPointReal));
			gICP.MFC8.actflow:=REAL_TO_UDINT(gICP.MFC8.actflowFloat);
			RETURN;
		END_IF
		t1(IN:=TRUE,PT:=T#200MS);
		IF t1.Q THEN
			gICP.MFC8.connectedCount:=gICP.MFC8.connectedCount+1;
			IF gICP.MFC8.connectedCount>10 THEN
				gICP.MFC8.connectedCount:=0;
				gICP.MFC8.connected:=FALSE;
				loopReadStep:=loopReadStep+10;
			ELSE
				loopReadStep:=loopReadStep+10;
			END_IF
			t1(IN:=FALSE);
		END_IF
	240:
		t1(IN:=TRUE,PT:=UDINT_TO_TIME(loopReadIntervalTime));
		IF t1.Q THEN
			loopReadStep:=loopReadStep+10;
			t1(IN:=FALSE);
		END_IF
	250:
		IF NOT gMFCStopLoopRead THEN
			Interface_Read(9);
			t1(IN:=FALSE);
			loopReadStep:=loopReadStep+10;
		ELSE
			loopReadStep:=5000;
		END_IF
	260:
		IF readDone THEN
			loopReadStep:=loopReadStep+10;
			gICP.MFC9.connected:=TRUE;
			gICP.MFC9.connectedCount:=0;
			t1(IN:=FALSE);
			gICP.MFC9.actflowFloat:=ReadLLimit(LREAL_TO_REAL(readPointReal));
			gICP.MFC9.actflow:=REAL_TO_UDINT(gICP.MFC9.actflowFloat);
			RETURN;
		END_IF
		t1(IN:=TRUE,PT:=T#200MS);
		IF t1.Q THEN
			gICP.MFC9.connectedCount:=gICP.MFC9.connectedCount+1;
			IF gICP.MFC9.connectedCount>10 THEN
				gICP.MFC9.connectedCount:=0;
				gICP.MFC9.connected:=FALSE;
				loopReadStep:=loopReadStep+10;
			ELSE
				loopReadStep:=loopReadStep+10;
			END_IF
			t1(IN:=FALSE);
		END_IF
	270:
		t1(IN:=TRUE,PT:=UDINT_TO_TIME(loopReadIntervalTime));
		IF t1.Q THEN
			loopReadStep:=loopReadStep+10;
			t1(IN:=FALSE);
		END_IF
	280:
		loopReadStep:=5000;
	5000:
		loopReadStep:=0;
END_CASE
END_ACTION

ACTION ACT_Read:
CASE readflowStep OF
	0:
	IF readExcute THEN
		readExcute:=FALSE;
		IF NOT serialBusy AND NOT readBusy AND NOT setBusy THEN
			readflowStep:=90;
			readBusy:=TRUE;
			readError:=FALSE;
			readDone:=FALSE;
		END_IF
	END_IF
	TimerReadPreset(IN:= FALSE);
	;
	
	90:
		readflowStep:=110;
		Read_Flow();
	100:
		;
	110:
		readPointStr:='';
		IF RcvDataFlag THEN
			readsetStarIndex:=FIND(arr_RcvDataString,'@');
			readsetPointStarIndex:=FIND(arr_RcvDataString,'$02');
			readsetPointEndIndex:=FIND(arr_RcvDataString,'$03');
			readIDStr:=MID(arr_RcvDataString,readsetPointStarIndex-readsetStarIndex-1,readsetStarIndex+1);
			readPointStr:=MID(arr_RcvDataString,readsetPointEndIndex-readsetPointStarIndex-1,readsetPointStarIndex+1);
			// readflowStep:=readflowStep+10;
			readPointInt:=STRING_TO_UDINT(readPointStr);
			readPointReal:=STRING_TO_LREAL(readPointStr);
			readIDInt:=STRING_TO_UDINT(readIDStr);
			readID:=(readIDInt=serialSlaveID);
			readflowStep:=5000;
			RETURN;
		END_IF
		TimerReadPreset(IN:= NOT TimerReadPreset.q, PT:=T#200MS);
		IF TimerReadPreset.Q THEN
			readflowStep:=6000;
			TimerReadPreset(IN:= FALSE);
			RETURN;
		END_IF
//	120:
//		readPointInt:=STRING_TO_UDINT(readPointStr);
//		readPointReal:=STRING_TO_LREAL(readPointStr);
//		readflowStep:=1000;
//	1000:
//		TimerReadPreset(IN:= NOT TimerReadPreset.q, PT:=T#00MS);
//		IF TimerReadPreset.Q THEN
//			readflowStep:=5000;
//			TimerReadPreset(IN:= FALSE);
//			// sendstr:='';
//		END_IF
	;
	5000://done
		readBusy:=FALSE;
		readflowStep:=0;
		readError:=FALSE;
		readDone:=TRUE;
	;
	6000://error
		readBusy:=FALSE;
		readflowStep:=0;
		readError:=TRUE;
		readDone:=FALSE;
	;
	
END_CASE
END_ACTION

ACTION ACT_Send:

CASE serialStep OF
	0:
	IF serialExcute THEN
		serialExcute:=FALSE;
		IF NOT serialBusy THEN
			serialStep:=90;
			serialBusy:=TRUE;
			serialDone:=FALSE;
			serialError:=FALSE;
			serialTimeOut:=FALSE;
			serialRecError:=FALSE;
		END_IF
	END_IF
	Timer1(IN:= FALSE);
	;
	
	90:
		arr_SendData:=sendbyte;
		serialStep:=100;
	100:
		send1(
			pSendData:= ADR(arr_SendData), 
			Length:= sendLenght, 
			Busy=> , 
			Error=> , 
			TXbuffer:= gTxBuffer_MFC);
		serialStep:=serialStep+10;
	110:
		Timer1(IN:= NOT timer1.q, PT:=T#10MS);
		IF Timer1.Q THEN
			serialStep:=serialStep+10;
			Timer1(IN:= FALSE);
		END_IF
	120:
		Timer1(IN:= NOT timer1.q, PT:=T#500MS);
		IF Timer1.Q THEN
			serialStep:=6000;
			Timer1(IN:= FALSE);
			serialTimeOut:=TRUE;
			RETURN;
		END_IF
		IF NOT send1.busy  THEN
			Timer1(IN:= FALSE);
			serialTimeOut:=FALSE;
			serialStep:=200;
		END_IF
		IF send1.Error <> COMERROR_NOERROR THEN
			serialRecError:=TRUE;
		END_IF
	200://数据处理
		serialStep:=serialStep+10;
	210:
		Timer1(IN:= NOT timer1.q, PT:=T#10MS);
		IF Timer1.Q THEN
			serialStep:=serialStep+10;
			Timer1(IN:= FALSE);
		END_IF
	220:
		//数据转换
		Timer1(IN:= FALSE);
		serialStep:=1000;
	
	1000:
		Timer1(IN:= NOT timer1.q, PT:=T#50MS);
		IF Timer1.Q THEN
			serialStep:=5000;
			Timer1(IN:= FALSE);
			// sendstr:='';
			serialTimeOut:=FALSE;
		END_IF
	;
	5000://done
		serialBusy:=FALSE;
		serialDone:=TRUE;
		serialError:=FALSE;
		serialStep:=0;
	;
	6000://error
		serialBusy:=FALSE;
		serialDone:=FALSE;
		serialError:=TRUE;
		serialStep:=0;
	;
	
END_CASE
END_ACTION

ACTION ACT_Set:
CASE setPresetStep OF
	0:
	IF setExcute THEN
		IF NOT serialBusy AND NOT setBusy THEN
			setExcute:=FALSE;
			setPresetStep:=90;
			setBusy:=TRUE;
			setError:=FALSE;
			setDone:=FALSE;
		END_IF
	END_IF
	TimerSetPreset(IN:= FALSE);
	;
	
	90:
		IF NOT FuncModule_RS485_MFC.readBusy AND FuncModule_RS485_MFC.loopReadStep<10 THEN
			Set_Flow(setPoint);
			setPresetStep:=100;
		END_IF
	100:
		TimerSetPreset(IN:= NOT TimerSetPreset.q, PT:=T#0MS);
		IF TimerSetPreset.Q THEN
			setPresetStep:=setPresetStep+10;
			TimerSetPreset(IN:= FALSE);
		END_IF
	110:
		IF RcvDataFlag THEN
			setPresetStep:=setPresetStep+10;
		END_IF
		TimerSetPreset(IN:= NOT TimerSetPreset.q, PT:=T#1000MS);
		IF TimerSetPreset.Q THEN
			setPresetStep:=6000;
			TimerSetPreset(IN:= FALSE);
			RETURN;
		END_IF
	120:
		IF FIND(arr_RcvDataString,'OK')>0 THEN
			//setPresetStep:=setPresetStep+10;
			setPresetStep:=5000;
		ELSE
			setPresetStep:=6000;
		END_IF
	130:
		setPresetStep:=setPresetStep+10;
		setBusy:=TRUE;
		TimerSetPreset(IN:= FALSE);
	140:
		arr_RcvDataString:='';
		Read_SetFlow();
		setPresetStep:=setPresetStep+10;
	150:
		readsetPointStr:='';
		IF RcvDataFlag THEN
			readsetPointStarIndex:=FIND(arr_RcvDataString,'$02');
			readsetPointEndIndex:=FIND(arr_RcvDataString,'$03');
			readsetPointStr:=MID(arr_RcvDataString,readsetPointEndIndex-readsetPointStarIndex-1,readsetPointStarIndex+1);
			setPresetStep:=setPresetStep+10;
		END_IF
		TimerSetPreset(IN:= NOT TimerSetPreset.q, PT:=T#1000MS);
		IF TimerSetPreset.Q THEN
			setPresetStep:=6000;
			TimerSetPreset(IN:= FALSE);
			RETURN;
		END_IF
	160:
		IF (STRING_TO_UDINT(readsetPointStr)<>setPoint) THEN
			setPresetStep:=6000;
		ELSE
			setPresetStep:=1000;
		END_IF
	
	1000:
		TimerSetPreset(IN:= NOT TimerSetPreset.q, PT:=T#50MS);
		IF TimerSetPreset.Q THEN
			setPresetStep:=5000;
			TimerSetPreset(IN:= FALSE);
			// sendstr:='';
		END_IF
	;
	5000://done
		setBusy:=FALSE;
		setPresetStep:=0;
		setError:=FALSE;
		setDone:=TRUE;
	;
	6000://error
		setBusy:=FALSE;
		setPresetStep:=0;
		setError:=TRUE;
		setDone:=FALSE;
	;
	
END_CASE
END_ACTION

METHOD CalASII_Byte : UDINT
VAR_INPUT
	date1:UDINT;
END_VAR
IF date1=10 THEN
	CalASII_Byte:=41;
END_IF
IF date1=11 THEN
	CalASII_Byte:=42;
END_IF
IF date1=12 THEN
	CalASII_Byte:=43;
END_IF
IF date1=13 THEN
	CalASII_Byte:=44;
END_IF
IF date1=14 THEN
	CalASII_Byte:=45;
END_IF
IF date1=15 THEN
	CalASII_Byte:=46;
END_IF
IF date1<10 THEN
	CalASII_Byte:=date1+30;
END_IF
IF date1>15 THEN
	CalASII_Byte:=date1+30;
END_IF
END_METHOD

METHOD Interface_Read : BOOL
VAR_INPUT
	sID:UDINT;
END_VAR
serialSlaveID:=sID;
readExcute:=TRUE;
END_METHOD

METHOD Interface_Set : BOOL
VAR_INPUT
	_sID:UDINT;
	_setPoint:UDINT;
END_VAR
serialSlaveID:=_sID;
setPoint:=_setPoint;
setExcute:=TRUE;
END_METHOD

METHOD Read_Flow : BOOL
VAR_INPUT

END_VAR
VAR
	sumq:UDINT;
	mod128:UDINT;
	intTemp:INT;
END_VAR
sendLenght:=9;
sendbyte[1]:=16#40;
sendbyte[2]:=UDINT_TO_BYTE((serialSlaveID/10)+48);// 48十进制转换成16进制为30；事实上是加30
sendbyte[3]:=UDINT_TO_BYTE((serialSlaveID MOD 10)+48);
sendbyte[4]:=16#02;
sendbyte[5]:=16#52;
sendbyte[6]:=16#46;
sendbyte[7]:=16#56;
sendbyte[8]:=16#03;
sumq:=0;
FOR intTemp:=5 TO UINT_TO_INT(sendLenght)-1 DO
	sumq:=sumq+sendbyte[intTemp];
END_FOR
mod128:=sumq MOD 128;
sendbyte[9]:=UDINT_TO_BYTE(mod128);
serialExcute:=TRUE;
END_METHOD

METHOD Read_SetFlow : BOOL
VAR_INPUT
END_VAR
VAR
	sumq:UDINT;
	mod128:UDINT;
	intTemp:INT;
END_VAR
sendLenght:=9;
sendbyte[1]:=16#40;
sendbyte[2]:=UDINT_TO_BYTE((serialSlaveID/10)+48);// 48十进制转换成16进制为30；事实上是加30
sendbyte[3]:=UDINT_TO_BYTE((serialSlaveID MOD 10)+48);
sendbyte[4]:=16#02;
sendbyte[5]:=16#52;
sendbyte[6]:=16#46;
sendbyte[7]:=16#43;
sendbyte[8]:=16#03;
sumq:=0;
FOR intTemp:=5 TO UINT_TO_INT(sendLenght)-1 DO
	sumq:=sumq+sendbyte[intTemp];
END_FOR
mod128:=sumq MOD 128;
sendbyte[9]:=UDINT_TO_BYTE(mod128);
serialExcute:=TRUE;
END_METHOD

METHOD ReadLLimit : REAL
VAR_INPUT
	input:REAL;
END_VAR
VAR_OUTPUT
END_VAR
VAR
	LLimit:REAL:=0;
END_VAR
IF input<LLimit THEN
	ReadLLimit:=LLimit;
ELSE
	ReadLLimit:=input;
END_IF
END_METHOD

METHOD Set_Flow : BOOL
VAR_INPUT
	flow:UDINT;
END_VAR
VAR
	sumq:UDINT;
	mod128:UDINT;
	intTemp:INT;
END_VAR
sendLenght:=14;
sendbyte[1]:=16#40;
sendbyte[2]:=UDINT_TO_BYTE((serialSlaveID/10)+48);// 48十进制转换成16进制为30；事实上是加30
sendbyte[3]:=UDINT_TO_BYTE((serialSlaveID MOD 10)+48);
sendbyte[4]:=16#02;
sendbyte[5]:=16#41;
sendbyte[6]:=16#46;
sendbyte[7]:=16#43;
sendbyte[8]:=UDINT_TO_BYTE((flow/100)+48);
IF sendbyte[8]>30 THEN
	sendbyte[9]:=UDINT_TO_BYTE((flow/10 MOD 10)+48);
ELSE
	sendbyte[9]:=UDINT_TO_BYTE((flow/10)+48);
END_IF
sendbyte[10]:=UDINT_TO_BYTE((flow MOD 10)+48);
sendbyte[11]:=16#2C;
sendbyte[12]:=16#42;
sendbyte[13]:=16#03;
sumq:=0;
FOR intTemp:=5 TO 13 DO
	sumq:=sumq+sendbyte[intTemp];
END_FOR
mod128:=sumq MOD 128;
sendbyte[14]:=UDINT_TO_BYTE(mod128);
serialExcute:=TRUE;
END_METHOD

END_PROGRAM

// ---- POUs/BaseModule/ActionModule/TMPModule/TMPModule.TcPOU
(*
--报错编号0: 无报错
--报错编号1: openend Error
--报错编号2: closeract Error
*)
FUNCTION_BLOCK TMPModule
VAR_IN_OUT
	WarmHMI					:WARMStruct;
	NoteHMI					:NoteStruct;
	operatorLog				:printLogModule_EX;
END_VAR
VAR_INPUT
	HMIItf						:TMPHMIStruts;//每个分子泵对象都关联了一个HMI
	TMPType						:TMPType:=TMPType_Default;//设置分子泵的类型
	real_TimeMonitor			:BOOL:=TRUE;//实时状态检测
	real_TimeMonitorClose		:BOOL:=FALSE;//实时状态检测关机
	runTime						: LINT;// 运行时间
	
	open						:BOOL:=FALSE;//启动触发信号
	openCondition				:BOOL:=TRUE;//启动条件
	close						:BOOL:=FALSE;//停止触发信号
	closeCondition				:BOOL:=TRUE;//停止条件
	reset						:BOOL:=FALSE;//复位信号
	stop						:BOOL:=FALSE;//停止信号
	power						:BOOL:=TRUE;//分子泵动作后是否关闭继电器得电状态, TRUE--保持得电,FALSE--断开得电
	enable						:BOOL:=TRUE;//分子泵禁用条件
	//ctrlMode					:ControlMode:=ControlMode.eManualCtrMode;//eManualCtrMode or eAutoCtrMode
	hmiEN						:BOOL:=TRUE;//HMI 启用条件
	serialExcute				:BOOL;// RS485开始一次参数读取
	
	errorDelayTime				:TIME:=T#5000MS;//分子泵感应器感应超时
	
	ACCMaxtime					:TIME:=T#3600S;// 分子泵加速最大时间
	DCCMaxtime					:TIME:=T#3600S;// 分子泵减速最大时间
	
	doneDelayTimeShortopenend	:TIME:=T#100MS;//分子泵启动感应到位延时_伸出
	doneDelayTimeShortcloseract	:TIME:=T#50MS;//分子泵感应到位延时_收回
	doneDelayTimeLongopenend	:TIME:=T#500MS;//无分子泵感应到位延时_伸出
	doneDelayTimeLongcloseract	:TIME:=T#50MS;//无分子泵感应到位延时_收回
	errorID						:UDINT:=0;//分子泵错误报警分配的起始ID
	nameTXT						:STRING(255):='';//分子泵名字
	
	AccAprSw					:BOOL:=FALSE;// 分子泵加速启动信号,需要链接到实际的IO点
	NormalAprSw					:BOOL:=FALSE;// 分子泵匀速感应器信号,需要链接到实际的IO点
	DccAprSw					:BOOL:=FALSE;// 分子泵减速感应器信号,需要链接到实际的IO点
	AlmAprSw					:BOOL:=FALSE;// 分子泵报警感应器信号,需要链接到实际的IO点
	ErrorAprSw					:BOOL:=FALSE;// 分子泵报错感应器信号,需要链接到实际的IO点
	enableOpenAprSw				:BOOL:=TRUE;// 启用启动感应器,针对只有一个传感器的分子泵
	enableCloseAprSw			:BOOL:=TRUE;// 启用停止感应器,针对只有一个传感器的分子泵
	
	mainPower					:BOOL;// 分子泵主电源
	temperature					:REAL;//分子泵温度
	current						:REAL;//分子泵电流
	speed						:REAL;//分子泵转速
	serialSlaveID				:UINT;// 分子泵ID
	serialError					:BOOL;// 分子泵通讯错误
	noteWTXT_open				:WSTRING(255):="";//分子泵打开动作NoteTXT 中文
	noteWTXT_close				:WSTRING(255):="";//分子泵关闭动作NoteTXT 中文
END_VAR
VAR_OUTPUT
	note_open				:BOOL;// 开条件不满足提示
	note_close				:BOOL;// 关条件不满足提示
	openRelay				:BOOL:=FALSE;// 分子泵启动执行继电器,需要链接到实际的IO点
	closeRelay				:BOOL:=FALSE;// 分子泵停止执行继电器,需要链接到实际的IO点
	resetRelay				:BOOL:=FALSE;// 分子泵复位执行继电器,需要链接到实际的IO点
	
	busy					:BOOL;//分子泵动作Busy状态
	openbusy				:BOOL;// 分子泵开动作Busy状态
	closebusy				:BOOL;// 分子泵关动作Busy状态
	resetbusy				:BOOL;// 分子泵关动作Busy状态
	done					:BOOL;//分子泵动作Done状态
	opendone					:BOOL;//分子泵动作伸出完成
	closedone					:BOOL;//分子泵动作收回完成
	resetdone					:BOOL;//分子泵动作收回完成
	error					:BOOL;//分子泵动作error状态
	errID					:UDINT;//分子泵动作errID
	errTXT					:STRING(255):='';//分子泵动作errTXT
	errWTXT					:WSTRING(255):="";//分子泵动作errTXT 中文
END_VAR
	
VAR	
	resetflag:BOOL;
	runTON			: TON;
	openErrorDelayTon		:Ton;
	openDoneDelayTon			:Ton;
	closeErrorDelayTon		:Ton;
	closeDoneDelayTon			:Ton;
	
	extendTrigRAlc			:R_Trig;//上升沿触发
	runTimeClearR			:R_Trig;//上升沿触发
	
	singleControlR			:R_Trig;//上升沿触发
	singleControlF			:F_Trig;//上升沿触发
	
	
	openendTrigRAlc			:R_Trig;//上升沿触发
	
	openendTrigR1			:R_Trig;//上升沿触发
	openendTrigR1_Aiko		:R_Trig;//上升沿触发
	closeractTrigR1			:R_Trig;//上升沿触发
	resetTrigR1				:R_Trig;//上升沿触发
	stopTrigR1				:R_Trig;//上升沿触发
	powerTrigR1				:R_Trig;//上升沿触发
	
	openStep				:UINT:=0;
	closeStep				:UINT:=0;
	errorStep				:UINT:=0;
	
	resetRelayTON			:TON;
	resetRecoverTON			:TON;
	resetRelayTONTime		:TIME:=T#0.5S;
	resetRecoverTime		:TIME:=T#1S;
	
	notBusyMonitorDelayTon:TON;//动作不切换时，延迟检测
	notBusyMonitorDelayTime:TIME:=T#2S;//动作不切换延迟检测时间
	firstPower			    :BOOL:=TRUE;//首次上电标志位
	
	AccFTrig:F_TRIG;//检测加速信号下降延
	NormalRTrig:R_TRIG;//匀速上升沿
	DccFTrig:F_TRIG;// 检测减速信号下降延
	noteTON_P:tON;            // 操作提示标志位延时继电器
	noteTON_N:tON;            // 操作提示标志位延时继电器
	noteRTrig_P:R_TRIG;          // 操作提示
	noteRTrig_N:R_TRIG;          // 操作提示
	powerTon:TON;
	extRealayRtrig:R_TRIG;
	retRealayRtrig:R_TRIG;
END_VAR

Init_ACT();
Error_ACT();
Open_ACT();
Close_ACT();
Reset_ACT();
Error_ACT();

(*
触发缩回动作，成功触发返回TRUE，触发失败返回FALSE
*)
METHOD Act_Close : BOOL
VAR_INPUT
END_VAR
IF enable AND closeCondition THEN// AND NOT busy
	Act_Close:=close:=TRUE;
ELSE
	Act_Close:=FALSE;
END_IF
END_METHOD

(*
触发伸出动作，成功触发返回TRUE，触发失败返回FALSE
*)
METHOD Act_Open : BOOL
VAR_INPUT
END_VAR
IF enable AND openCondition THEN// AND NOT busy
	Act_Open:=open:=TRUE;
ELSE
	Act_Open:=FALSE;
END_IF
END_METHOD

(*
触发复位报警动作，成功触发返回TRUE，触发失败返回FALSE
*)
METHOD Act_Reset : BOOL
VAR_INPUT
END_VAR
Act_Reset:=reset:=TRUE;
END_METHOD

(*
触发发送动作，成功触发返回TRUE，触发失败返回FALSE
*)
METHOD Act_SerialSend : BOOL
VAR_INPUT
END_VAR
IF TRUE THEN
	Act_SerialSend:=serialExcute:=TRUE;
ELSE
	Act_SerialSend:=FALSE;
END_IF
END_METHOD

(*
触发停止输出动作，成功触发返回TRUE，触发失败返回FALSE
*)
METHOD Act_Stop : BOOL
VAR_INPUT
END_VAR
Act_Stop:=stop:=TRUE;
END_METHOD

ACTION Close_ACT:
//分子泵--close 触发
IF close AND NOT closeCondition THEN
	note_open:=FALSE;
	note_close:=TRUE;
	NoteHMI.showFlag:=TRUE;
	NoteHMI.showText:='';
	NoteHMI.showText:=CONCAT(NoteHMI.showText,nameTXT);
	NoteHMI.showText:=CONCAT(NoteHMI.showText,' Close Condition Not Satisfied!');
	operatorLog.append(CONCAT(nameTXT,' Close Not Done '));
END_IF
IF close AND enable AND closeCondition AND closeStep<20 THEN// AND NOT busy
	note_open:=FALSE;
	note_close:=FALSE;
	busy:=TRUE;
	closebusy:=TRUE;
	openbusy:=FALSE;
	resetbusy:=FALSE;
	open:=FALSE;
	reset:=FALSE;
	resetdone:=FALSE;
	opendone:=FALSE;
	closedone:=FALSE;
	openStep:=0;
	closeStep:=10;
	closeStep:=10;
	gTBPStopLoopRead:=TRUE;
	FuncModule_RS232_TBP.Interface_Stop();
	FuncModule_RS232_TBP.startStep:=0;
	FuncModule_RS232_TBP.stopStep:=0;
	FuncModule_RS232_TBP.resetStep:=0;
	operatorLog.append(CONCAT(nameTXT,' Close Done '));
	//errorStep:=0;
END_IF
close:=FALSE;

CASE closeStep OF
0:
	//ready
	
10:
	IF FuncModule_RS232_TBP.loopReadStep<10 AND FuncModule_RS232_TBP.startStep<10 
	   AND FuncModule_RS232_TBP.resetStep<10 THEN
		closeErrorDelayTon(IN:=FALSE);
		closeDoneDelayTon(IN:=FALSE);
		closeRelay:=TRUE;
		openRelay:=FALSE;
		closeStep:=15;
	END_IF;
15:
	IF FuncModule_RS232_TBP.stopDone THEN
		closeStep:=20;
		gTBPStopLoopRead:=FALSE;
		RETURN;
	END_IF
	IF FuncModule_RS232_TBP.stopError THEN
		errorStep:=2;
		open:=FALSE;
		close:=FALSE;
		reset:=FALSE;
		openbusy:=FALSE;
		closebusy:=FALSE;
		resetbusy:=FALSE;
		closeStep:=60;
		gTBPStopLoopRead:=FALSE;
		RETURN;
	END_IF
20:
	IF NOT DccAprSw AND NOT openRelay AND NOT NormalAprSw AND NOT AccAprSw AND speed<5 THEN
		closeStep:=40;
	ELSE
		closeErrorDelayTon(IN:=(NOT DccAprSw AND enablecloseAprSw),PT:=errorDelayTime);
		IF closeErrorDelayTon.Q THEN
			//done:=FALSE;
			opendone:=FALSE;
			closedone:=FALSE;
			resetdone:=FALSE;
			errorStep:=2;
			closebusy:=FALSE;
			openbusy:=FALSE;
			resetbusy:=FALSE;
			closeStep:=60;
			RETURN;
		END_IF
		IF enablecloseAprSw THEN
			closeDoneDelayTon(IN:=DccAprSw,PT:=doneDelayTimeShortcloseract);
		END_IF
		IF closeDoneDelayTon.Q OR (DccAprSw AND NOT openRelay AND NOT NormalAprSw AND NOT AccAprSw)  THEN
			closeErrorDelayTon(IN:=FALSE);
			closeDoneDelayTon(IN:=FALSE);
			closeStep:=30;
		END_IF
	END_IF
30:
	closeErrorDelayTon(IN:=DccAprSw,PT:=DCCMaxtime);
	IF closeErrorDelayTon.Q THEN
		//done:=FALSE;
		opendone:=FALSE;
		closedone:=FALSE;
		resetdone:=FALSE;
		closeStep:=60;
		openRelay:=FALSE;
		errorStep:=2;
		closebusy:=FALSE;
		openbusy:=FALSE;
		resetbusy:=FALSE;
		closeErrorDelayTon(IN:=FALSE);
	END_IF
	DccFTrig(CLK:=DccAprSw );
	IF DccFTrig.Q OR (NOT DccAprSw AND NOT openRelay AND NOT NormalAprSw AND NOT AccAprSw) THEN
		closeStep:=40;
		closeErrorDelayTon(IN:=FALSE);
	END_IF
40:
	IF NOT DccAprSw AND NOT NormalAprSw THEN
		IF NOT AccAprSw AND speed<5 THEN
			busy:=FALSE;
			closebusy:=FALSE;
			openbusy:=FALSE;
			resetbusy:=FALSE;
			//done:=TRUE;
			opendone:=FALSE;
			closedone:=TRUE;
			resetdone:=FALSE;
			errorStep:=0;
			closeStep:=50;
			IF NOT power (*AND NOT (CylinderType_Vacuum=cylinderType)*) THEN
				openRelay:=FALSE;
				closeRelay:=FALSE;
			END_IF
			closeRelay:=FALSE;
		ELSE
			busy:=FALSE;
			closebusy:=FALSE;
			openbusy:=FALSE;
			resetbusy:=FALSE;
			//done:=TRUE;
			opendone:=FALSE;
			closedone:=FALSE;
			resetdone:=FALSE;
			errorStep:=3;
			closebusy:=FALSE;
			openbusy:=FALSE;
			resetbusy:=FALSE;
			closeStep:=60;
		END_IF
	END_IF
END_CASE
END_ACTION

ACTION Error_ACT:
CASE errorStep OF
	0:
		error:=FALSE;
		errID:=0;
		errTXT:='';
 (*
	1:
		error:=TRUE;
		errID:=errorID+errorStep;
		errTXT:=CONCAT(STR1:=nameTXT,STR2:=' Extend Error!');
		errWTXT:=WCONCAT(STR1:=TO_WSTRING(nameTXT),STR2:=" 伸出(打开)错误");
	2:
		error:=TRUE;
		errID:=errorID+errorStep;
		errTXT:=CONCAT(STR1:=nameTXT,STR2:=' Retract Error!');
		errWTXT:=WCONCAT(STR1:=TO_WSTRING(nameTXT),STR2:=" 缩回(关闭)错误");
		*)
	1..6:
		error:=TRUE;
		errID:=getErrID(errorStep);
		errTXT:=getErrTXT(errorStep);
		errWTXT:=getErrWTXT(errorStep);
END_CASE
END_ACTION

METHOD Get_Done_Close : BOOL
VAR_INPUT
END_VAR
Get_Done_Close:=closedone;
END_METHOD

METHOD Get_Done_Open : BOOL
VAR_INPUT
END_VAR
Get_Done_Open:=opendone;
END_METHOD

METHOD getErrID : UDINT
VAR_INPUT
	errID					:UDINT;//取值范围1~2
END_VAR
VAR
	nErrID					:UDINT;
END_VAR
nErrID:=errorID+errID;

getErrID:=nErrID;
END_METHOD

METHOD getErrTXT : STRING(255)
VAR_INPUT
	errID					:UDINT;//取值范围1~2
END_VAR
VAR
	sErrTXT					:STRING(255);
END_VAR

CASE errID OF
	1:
		sErrTXT:=CONCAT(STR1:=nameTXT,STR2:=' Open Error!');
	2:
		sErrTXT:=CONCAT(STR1:=nameTXT,STR2:=' Close Error!');
	3:
		sErrTXT:=CONCAT(STR1:=nameTXT,STR2:=' NormalRun Error!');
	4:
		sErrTXT:=CONCAT(STR1:=nameTXT,STR2:=' CheckCondition Error!');
	5:
		sErrTXT:=CONCAT(STR1:=nameTXT,STR2:=' IO Fault!');
	6:
		sErrTXT:=CONCAT(STR1:=nameTXT,STR2:=' Communication Error!');
ELSE
	sErrTXT:=CONCAT(STR1:=nameTXT,STR2:='');
END_CASE
getErrTXT:=sErrTXT;
END_METHOD

METHOD getErrWTXT : WSTRING(255)
VAR_INPUT
	errID					:UDINT;//取值范围1~16
END_VAR
VAR
	sErrTXT					:WSTRING(255);
END_VAR

CASE errID OF
	1:
		sErrTXT:=WCONCAT(STR1:=TO_WSTRING(nameTXT),STR2:=" 分子泵启动错误");
	2:
		sErrTXT:=WCONCAT(STR1:=TO_WSTRING(nameTXT),STR2:=" 分子泵停止错误");
	3:
		sErrTXT:=WCONCAT(STR1:=TO_WSTRING(nameTXT),STR2:=" 分子泵正常运行出现异常情况");
	4:
		sErrTXT:=WCONCAT(STR1:=TO_WSTRING(nameTXT),STR2:=" 检测到条件异常，关机处理");
	5:
		sErrTXT:=WCONCAT(STR1:=TO_WSTRING(nameTXT),STR2:=" 分子泵IO报错");
	6:
		sErrTXT:=WCONCAT(STR1:=TO_WSTRING(nameTXT),STR2:=" 分子泵通讯异常");
ELSE
	sErrTXT:=WCONCAT(STR1:=TO_WSTRING(nameTXT),STR2:="");
END_CASE
getErrWTXT:=sErrTXT;
END_METHOD

ACTION Init_ACT:
done:=(opendone OR closedone);
powerTon(IN:=mainPower,PT:=T#10S);
IF AlmAprSw AND powerTon.Q THEN
	errorStep:=5;
END_IF
IF FuncModule_RS232_TBP.serialTimeoutError THEN
	errorStep:=6;
END_IF
error:=error OR serialError OR NOT mainPower OR AlmAprSw;
InitHMI_ACT();
manualCtrl_ACT();
IF (error OR AlmAprSw OR ErrorAprSw) AND openRelay THEN
	stop:=TRUE;
	busy:=FALSE;
	openRelay:=FALSE;
END_IF

noteTON_P(IN:=note_open,PT:=T#0.1S);
noteRTrig_P(CLK:=noteTON_P.Q);
IF noteRTrig_P.Q THEN
//	gLog_Note.append_EX(noteWTXT_Open);
END_IF
noteTON_N(IN:=note_close,PT:=T#0.1S);
noteRTrig_N(CLK:=noteTON_N.Q);
IF noteRTrig_N.Q THEN
//	gLog_Note.append_EX(noteWTXT_close);
END_IF
extRealayRtrig(CLK:=openRelay);
IF extRealayRtrig.Q THEN
	HMIItf.singleControl:=TRUE;
END_IF
retRealayRtrig(CLK:=NOT openRelay);
IF retRealayRtrig.Q THEN
	HMIItf.singleControl:=FALSE;
END_IF
IF NOT gICP.TruboPumNoRotation AND FuncModule_RS232_TBP.serialConnected AND firstPower AND NOT HMIItf.singleControl THEN
	HMIItf.singleControl:=TRUE;
	openRelay:=TRUE;
	firstPower:=FALSE;
END_IF
END_ACTION

ACTION InitHMI_ACT:
HMIItf.AccAprSw:=AccAprSw;
HMIItf.NormalAprSw:=NormalAprSw;
HMIItf.AlmAprSw:=AlmAprSw;
HMIItf.DccAprSw:=DccAprSw;
HMIItf.ErrorAprSw:=ErrorAprSw;

HMIItf.temperature:=temperature;
HMIItf.current:=current;
HMIItf.speed:=speed;

HMIItf.enableOpen:=enableOpenAprSw;
HMIItf.enableClose:=enableCloseAprSw;
HMIItf.HMIEnable:=hmiEN;
HMIItf.enable:=enable;
HMIItf.done:=done;
HMIItf.busy:=busy;
HMIItf.error:=error;
HMIItf.errID:=UDINT_TO_DINT(errID);
HMIItf.errTXT:=errTXT;
HMIItf.openRelay:=openRelay;
HMIItf.resetRelay:=resetRelay;

HMIItf.power:=power;
HMIItf.nameTXT:=nameTXT;

HMIItf.runTime:=runTime;
HMIItf.opencondition:=openCondition;
HMIItf.closecondition:=closeCondition;
END_ACTION

ACTION ManualCtrl_ACT:
//HMI手动控制
//IF ctrlMode=eManualCtrMode THEN
IF hmiEN THEN
	singleControlR(CLK:=HMIItf.singleControltemp);
	openendTrigR1_Aiko(CLK:=HMIItf.bopen);
	IF (openendTrigR1_Aiko.Q OR (HMIItf.singleControltemp AND NOT HMIItf.singleControl)) THEN
		WarmHMI.showText:='';
		WarmHMI.showFlag:=TRUE;
		WarmHMI.showText:=CONCAT(WarmHMI.showText,'Are you sure you want to Open the ');
		WarmHMI.showText:=CONCAT(WarmHMI.showText,nameTXT);
		WarmHMI.showText:=CONCAT(WarmHMI.showText,' ?');
	END_IF
	IF WarmHMI.bOK AND NOT WarmHMI.showFlag AND FIND(WarmHMI.showText,nameTXT)>0 AND FIND(WarmHMI.showText,'Open')>0 THEN
		open:=TRUE;
		close:=FALSE;
		IF NOT HMIItf.singleControl AND openCondition THEN
			HMIItf.singleControl:=NOT HMIItf.singleControl;
		END_IF
		operatorLog.append(CONCAT(nameTXT,' Open'));
		WarmHMI.showText:='';
		WarmHMI.bOK:=FALSE;
		WarmHMI.showText:='';
	END_IF
	IF WarmHMI.bNO AND NOT WarmHMI.showFlag AND FIND(WarmHMI.showText,nameTXT)>0 AND FIND(WarmHMI.showText,'Open')>0 THEN
		WarmHMI.bNO:=FALSE;
		WarmHMI.showText:='';
	END_IF
	
	IF (openendTrigR1_Aiko.Q OR (HMIItf.singleControltemp AND HMIItf.singleControl)) THEN
		WarmHMI.showText:='';
		WarmHMI.showFlag:=TRUE;
		WarmHMI.showText:=CONCAT(WarmHMI.showText,'Are you sure you want to Close the ');
		WarmHMI.showText:=CONCAT(WarmHMI.showText,nameTXT);
		WarmHMI.showText:=CONCAT(WarmHMI.showText,' ?');
	END_IF
	IF WarmHMI.bOK AND NOT WarmHMI.showFlag AND FIND(WarmHMI.showText,nameTXT)>0 AND FIND(WarmHMI.showText,'Close')>0 THEN
		close:=TRUE;
		operatorLog.append(CONCAT(nameTXT,' Close'));
		open:=FALSE;
		IF HMIItf.singleControl AND closeCondition THEN
			HMIItf.singleControl:=NOT HMIItf.singleControl;
		END_IF
		WarmHMI.showText:='';
		WarmHMI.bOK:=FALSE;
		WarmHMI.showText:='';
	END_IF
	IF WarmHMI.bNO AND NOT WarmHMI.showFlag AND FIND(WarmHMI.showText,nameTXT)>0 AND FIND(WarmHMI.showText,'Close')>0 THEN
		WarmHMI.bNO:=FALSE;
		WarmHMI.showText:='';
	END_IF
	
	openendTrigR1(CLK:=HMIItf.open);
	IF openendTrigR1.Q THEN// AND NOT busy
		open:=TRUE;
	END_IF
	
	closeractTrigR1(CLK:=HMIItf.close);
	IF closeractTrigR1.Q THEN// AND NOT busy
		close:=TRUE;
	END_IF
	
	resetTrigR1(CLK:=HMIItf.reset);
	IF resetTrigR1.Q THEN// AND NOT busy
		reset:=TRUE;
	END_IF
	
	stopTrigR1(CLK:=HMIItf.stop);
	IF stopTrigR1.Q THEN// AND NOT busy
		stop:=TRUE;
	END_IF
	
	powerTrigR1(CLK:=HMIItf.power);
	IF powerTrigR1.Q THEN// AND NOT busy
		IF power THEN
			power:=FALSE;
		ELSE
			power:=TRUE;
		END_IF
	END_IF
	
END_IF
END_ACTION

ACTION Open_ACT:
//分子泵伸出--open 触发
IF open AND NOT openCondition THEN
	note_open:=TRUE;
	note_close:=FALSE;
	NoteHMI.showFlag:=TRUE;
	NoteHMI.showText:='';
	NoteHMI.showText:=CONCAT(NoteHMI.showText,nameTXT);
	NoteHMI.showText:=CONCAT(NoteHMI.showText,' Open Condition Not Satisfied!');
	operatorLog.append(CONCAT(nameTXT,' Open Not Done '));
END_IF
IF open AND enable AND openCondition AND NOT AlmAprSw AND NOT ErrorAprSw AND NOT openbusy AND mainPower AND NOT resetRelay THEN// AND NOT busy
	note_open:=FALSE;
	note_close:=FALSE;
	busy:=TRUE;
	closebusy:=FALSE;
	resetbusy:=FALSE;
	openbusy:=TRUE;
	close:=FALSE;
	open:=FALSE;
	reset:=FALSE;
	done:=FALSE;
	opendone:=FALSE;
	closedone:=FALSE;
	resetdone:=FALSE;
	openStep:=10;
	closeStep:=0;
	gTBPStopLoopRead:=TRUE;
	FuncModule_RS232_TBP.startStep:=0;
	FuncModule_RS232_TBP.stopStep:=0;
	FuncModule_RS232_TBP.resetStep:=0;
	operatorLog.append(CONCAT(nameTXT,' Open Done '));
END_IF
open:=FALSE;
runTimeClearR(CLK:=HMIItf.runTimeClear);
runTON(IN:=NOT error AND openRelay AND(AccAprSw OR DccAprSw OR NormalAprSw) AND NOT runTON.Q, PT:=T#3600S);// 1小时计数一次,启动，无报错，且全速
IF runTON.Q AND runTime<999999999999999 AND NOT runTimeClearR.Q THEN
	runTime:=runTime+1;
END_IF
IF runTimeClearR.Q THEN
	runTime:=0;
END_IF
//IF NOT openRelay AND NOT AccAprSw AND NOT DccAprSw AND NOT NormalAprSw THEN// 计数清零
//	runTime:=0;
//END_IF

CASE openStep OF
0:
	//ready
	runTON(IN:=FALSE);
10:
	IF FuncModule_RS232_TBP.loopReadStep<10
	   AND FuncModule_RS232_TBP.stopStep<10 AND FuncModule_RS232_TBP.resetStep<10 THEN
		openErrorDelayTon(IN:=FALSE);
		openDoneDelayTon(IN:=FALSE);
		openStep:=15;
		openRelay:=TRUE;
		FuncModule_RS232_TBP.Interface_Start();
		openbusy:=FALSE;
		closebusy:=FALSE;
		resetbusy:=FALSE;
		closeRelay:=FALSE;
	END_IF
15:
	IF FuncModule_RS232_TBP.startDone THEN
		openStep:=20;
		gTBPStopLoopRead:=FALSE;
		RETURN;
	END_IF
	IF FuncModule_RS232_TBP.startError THEN
		errorStep:=1;
		open:=FALSE;
		close:=FALSE;
		reset:=FALSE;
		openbusy:=FALSE;
		closebusy:=FALSE;
		resetbusy:=FALSE;
		openStep:=60;
		gTBPStopLoopRead:=FALSE;
		RETURN;
	END_IF
20:
	openErrorDelayTon(IN:=((NOT AccAprSw AND NOT NormalAprSw) AND enableopenAprSw),PT:=errorDelayTime);
	IF openErrorDelayTon.Q THEN
		//done:=FALSE;
		open:=FALSE;
		close:=FALSE;
		openbusy:=FALSE;
		resetbusy:=FALSE;
		closebusy:=FALSE;
		resetbusy:=FALSE;
		errorStep:=1;
		openStep:=60;
		RETURN;
	END_IF
	IF enableopenAprSw THEN
		openDoneDelayTon(IN:=(AccAprSw OR NormalAprSw),PT:=doneDelayTimeShortopenend);
	END_IF
	IF openDoneDelayTon.Q THEN
		openErrorDelayTon(IN:=FALSE);
		openDoneDelayTon(IN:=FALSE);
		openStep:=30;
	END_IF
	
	//状态实时检测
	IF NOT openCondition AND (NOT closedone OR openRelay) THEN//蝶阀单控，检测到开条件消失，强制关闭
		close:=TRUE;
		openRelay:=FALSE;
		HMIItf.singleControltemp:=FALSE;
		errorStep:=4;
		openbusy:=FALSE;
		closebusy:=FALSE;
		resetbusy:=FALSE;
		resetbusy:=FALSE;
		openStep:=60;
	END_IF
	IF (ErrorAprSw OR AlmAprSw) AND openRelay THEN//只要报错；启动线圈启动，强锁启动信号
		openRelay:=FALSE;
		HMIItf.singleControltemp:=FALSE;
		close:=TRUE;
		stop:=TRUE;
		openStep:=60;/////
		errorStep:=3;
		openbusy:=FALSE;
		closebusy:=FALSE;
		resetbusy:=FALSE;
	END_IF
30:
	openErrorDelayTon(IN:=AccAprSw OR NormalAprSw,PT:=ACCMaxtime);
	IF openErrorDelayTon.Q THEN
		//done:=FALSE;
		opendone:=FALSE;
		closedone:=FALSE;
		resetdone:=FALSE;
		openStep:=60;
		//openRelay:=FALSE;
		errorStep:=1;
		closebusy:=FALSE;
		openbusy:=FALSE;
		resetbusy:=FALSE;
		openErrorDelayTon(IN:=FALSE);
	END_IF
	AccFTrig(CLK:=AccAprSw);
	IF AccFTrig.Q OR NormalAprSw THEN
		openStep:=40;
		openErrorDelayTon(IN:=FALSE);
	END_IF
	//状态实时检测
	IF NOT openCondition AND (NOT closedone OR openRelay) THEN//蝶阀单控，检测到开条件消失，强制关闭
		close:=TRUE;
		openRelay:=FALSE;
		HMIItf.singleControltemp:=FALSE;
		errorStep:=4;
		openStep:=60;
		closebusy:=FALSE;
		openbusy:=FALSE;
		resetbusy:=FALSE;
	END_IF
	IF (ErrorAprSw OR AlmAprSw) AND openRelay THEN//只要报错；启动线圈启动，强锁启动信号
		openRelay:=FALSE;
		HMIItf.singleControltemp:=FALSE;
		close:=TRUE;
		stop:=TRUE;
		openStep:=60;/////
		errorStep:=3;
		closebusy:=FALSE;
		openbusy:=FALSE;
		resetbusy:=FALSE;
	END_IF
40:
	IF NormalAprSw THEN
		IF NOT DccAprSw AND NOT AccAprSw THEN
			busy:=FALSE;
			closebusy:=FALSE;
			openbusy:=FALSE;
			resetbusy:=FALSE;
			//done:=TRUE;
			opendone:=TRUE;
			closedone:=FALSE;
			resetdone:=FALSE;
			errorStep:=0;
			openStep:=50;
			IF NOT power (*AND NOT (CylinderType_Vacuum=cylinderType)*) THEN
				openRelay:=FALSE;
				HMIItf.singleControltemp:=FALSE;
				closeRelay:=FALSE;
			END_IF
		ELSE
			busy:=FALSE;
			closebusy:=FALSE;
			openbusy:=FALSE;
			resetbusy:=FALSE;
			//done:=TRUE;
			opendone:=FALSE;
			resetdone:=FALSE;
			closedone:=FALSE;
			errorStep:=3;
			openStep:=60;
		END_IF
	END_IF
50:
	IF real_TimeMonitor THEN
		//启动实时检测
		IF (enableOpenAprSw AND(NOT NormalAprSw)) AND openRelay THEN
			errorStep:=1;
			openRelay:=FALSE;
			HMIItf.singleControltemp:=FALSE;
			openStep:=60;
			closebusy:=FALSE;
			openbusy:=FALSE;
			resetbusy:=FALSE;
		END_IF
//		IF NOT openCondition AND (NOT closedone OR openRelay) THEN//蝶阀单控，检测到开条件消失，强制关闭
//			openRelay:=FALSE;
//			HMIItf.singleControltemp:=FALSE;
//			errorStep:=4;
//			openStep:=60;
//			closebusy:=FALSE;
//			openbusy:=FALSE;
//			resetbusy:=FALSE;
//		END_IF
		IF (ErrorAprSw OR AlmAprSw) AND openRelay THEN//只要报错；启动线圈启动，强锁启动信号
			openRelay:=FALSE;
			HMIItf.singleControltemp:=FALSE;
			stop:=TRUE;
			openStep:=60;/////
			errorStep:=3;
			closebusy:=FALSE;
			openbusy:=FALSE;
			resetbusy:=FALSE;
		END_IF
		IF real_TimeMonitorClose THEN
			openRelay:=FALSE;
			HMIItf.singleControltemp:=FALSE;
			stop:=TRUE;
			openStep:=60;/////
			errorStep:=4;
			closebusy:=FALSE;
			openbusy:=FALSE;
			resetbusy:=FALSE;
		END_IF
	END_IF
60:
	;//报错
END_CASE
END_ACTION

ACTION Reset_ACT:
IF reset THEN
	IF NOT power THEN
		openRelay:=FALSE;
		closeRelay:=FALSE;
	END_IF
	note_open:=FALSE;
	note_close:=FALSE;
	IF errorStep<>0 OR  AlmAprSw OR ErrorAprSw THEN
		openStep:=0;
		closeStep:=0;
		errorStep:=0;
		busy:=FALSE;
		resetRelay:=TRUE;
		gTBPStopLoopRead:=TRUE;
	END_IF
	reset:=FALSE;
	note_open:=FALSE;
	note_close:=FALSE;
END_IF
resetRelayTON(IN:=resetRelay AND FuncModule_RS232_TBP.loopReadStep=0, PT:=resetRelayTONTime);// 500MS 触发读写锁；
IF resetRelayTON.Q THEN
	openStep:=0;
	closeStep:=0;
	errorStep:=0;
	busy:=FALSE;
	resetRelay:=FALSE;
	FuncModule_RS232_TBP.Interface_Reset();
	resetflag:=TRUE;
END_IF
resetRecoverTON(IN:=resetflag , PT:=resetRecoverTime);// 1S后触发复位
IF resetRecoverTON.Q THEN
	resetflag:=FALSE;;
	gTBPStopLoopRead:=FALSE;
	resetRelay:=FALSE;
END_IF
IF stop THEN
	note_open:=FALSE;
	note_close:=FALSE;
	stop:=FALSE;
	openRelay:=FALSE;
	closeRelay:=FALSE;
	//无自锁检测说法，直接停
	openStep:=0;
	closeStep:=0;
	gTBPStopLoopRead:=TRUE;
	FuncModule_RS232_TBP.Interface_Stop();
END_IF
END_ACTION

ACTION VersionLog:
(*
版本: V1.0.0.0
说明:
	1. 首个版本
	2. 含普通分子泵\泵组类型的控制
	3. 可配置是否有到位信号, 以及到位稳定时间
(--------------------------------------------------)
新版本: V1.0.1.0
更新时间: 2019/11/20 19:00
更新说明:
	1. 优化编写方式
	2. 修改错误编码起始位，现改为从1开始
(--------------------------------------------------)
新版本: V1.0.1.1
更新时间: 2020/03/23 23:00
更新说明:
	1. 优化报错方式
	2. 增加伸出、缩回、复位和停止触发函数
(--------------------------------------------------)
新版本: V1.0.1.2
更新时间: 2020/04/22 09:50
更新说明:
	1. 增加中文报警输出
(--------------------------------------------------)
新版本: V1.0.1.3
更新时间: 2020/09/16
更新说明:
	1. 开放错误ID、错误文本信息获取接口
(--------------------------------------------------)
新版本: V1.0.1.4
更新时间: 2020/10/06
更新说明:
	1. 移除控制模式变量，增加HMI启用条件
	2. 增加外部获取伸出缩回完成信号接口函数
(--------------------------------------------------)
新版本: V1.0.1.5
更新时间: 2020/10/14
更新说明:
	1. 优化代码
(--------------------------------------------------)
新版本: V2.0.1.0
更新时间: 2023/11/17
更新说明:
	1. 分子泵控制独立
(--------------------------------------------------)


*)
END_ACTION

END_FUNCTION_BLOCK

// ---- POUs/BaseModule/Communication/FuncModule_RS232_TBP.TcPOU
PROGRAM FuncModule_RS232_TBP
VAR_IN_OUT
	
END_VAR
VAR_INPUT
	serialSlaveID				:UDINT:=1;// 从站节点号
	sendLenght					:UINT:=14;// 发送字节长度
	sendbyte					:ARRAY[1..20]			OF		BYTE;(*READ*)//发送数据
	timeout						:TIME:=T#100MS;// 超时时间
	setPoint					:UDINT;
	loopReadStep				:INT;
	loopReadExcute				:BOOL;
	loopReadIntervalTime		:UDINT:=0;
	
	startStep						:UINT;				//处理步数
	stopStep						:UINT;				//处理步数
	resetStep						:UINT;				//处理步数
END_VAR
VAR_OUTPUT
	serialBusy						:BOOL;
	startBusy						:BOOL;
	stopBusy						:BOOL;
	resetBusy						:BOOL;
	serialDone						:BOOL;
	startDone						:BOOL;
	stopDone						:BOOL;
	resetDone						:BOOL;
	serialError						:BOOL;
	startError						:BOOL;
	stopError						:BOOL;
	resetError						:BOOL;
	serialConnected					:BOOL;
	setBusy							:BOOL;// 设置参数时繁忙
	setError						:BOOL;
	setDone							:BOOL;
	readBusy						:BOOL;// 读取参数时繁忙
	readError						:BOOL;
	readDone						:BOOL;
	
	serialTimeoutError				:BOOL;
	
	noRotation:BOOL; // 静止
	brake:BOOL;		// 制动
	acc:BOOL;		// 加速
	atTagetSpeed:BOOL;// 全速
	alarm:BOOL;		 // 警告
	remote:BOOL;	 // 远程操作中 远程操作为1
	failure:BOOL;		// 报错
	rotationSpeed:UDINT;// 实时转速（HZ）
	tMSTemperature:REAL;// 温度
END_VAR
VAR
	serialExcute				:BOOL;// RS232开始一次参数读取
	startExcute					:BOOL;// RS232
	stopExcute					:BOOL;// RS232
	resetExcute					:BOOL;// RS232

	intTemp						:UDINT;
	
	realTemp						:REAL;
	loopToReadRatationTimes			:INT;
	prefix						:STRING:='';// 字符串头
	suffix						:STRING:= '';// 字符串尾
	readsetPointStarIndex				:INT;
	readsetPointEndIndex				:INT;
	readsetPointStr				:STRING;
	readPointStr				:STRING;
	readPointReal				:LREAL;
	readPointInt				:UDINT;
	//Byte方式
	send1:							SendData;
	receive1:						ReceiveData;
	Timer1:							TON;
	TimerStart:						TON;
	TimerStop:						TON;
	TimerReset:						TON;
	
	TimerStartTOut:						TON;
	TimerStopTOut:						TON;
	TimerResetTOut:						TON;
	TimerSetPreset:							TON;
	TimerReadPreset:							TON;
	t1:								TON;
	t2:								TON;
	timeoutResetTime				:TON;
	timeToNext						:TIME:=T#10MS;
	arr_SendData:					ARRAY[1..20]			OF		BYTE;(*READ*)//发送数据
	arr_SendDataTemp				:ARRAY[1..20]			OF		BYTE;(*READ*)//发送数据
	arr_RcvDataByte:				ARRAY[1..20]			OF		BYTE;;// 接收数据
	arr_RcvDataByteTemp:				ARRAY[1..20]			OF		BYTE;;// 接收数据
	arr_RcvDataByteClear:			ARRAY[1..20]			OF		BYTE;;// 清除接收数据
	RcvDataFlag:			BOOL;// 接收数据标志位
	serialStep						:UINT;				//处理步数
	serialTimeOut:BOOL;//接收数据超时
	serialTimeOutTimes:INT:=0;//接收数据超时次数
	serialRecError:BOOL;//接收数据错误
	reciveFtrig:F_TRIG;
	recTon:TON;
	againSendS3:TON;
	hexChars:ARRAY [0..15] OF STRING[1]:=['0','1','2','3','4','5','6','7','8','9','A','B','C','D','E','F'];
	loopreadConditionTON:TON;
END_VAR

(*
 *功能块的作用，把 TxBuffer 缓存区的数据经过 Process Data 的 ComOut 发送出去，
 *而把 ComIn 中的数据接收到 RxBuffer。引用这个功能块的程序执行周期越短，
 *数据交换的效率就越高，所以这段程序应该放在快速任务中作为 Backgroud 代码无条件执行。
*)
IF receive1.Error <> COMERROR_NOERROR THEN
	serialRecError:=TRUE;
END_IF
receive1(
	pPrefix:= , 
	LenPrefix:= , 
	pSuffix:= , 
	LenSuffix:= , 
	pReceiveData:= ADR(arr_RcvDataByteTemp), 
	SizeReceiveData:= 20, 
	Timeout:= timeout, //临时设置成10S调试用
	Reset:= , 
	DataReceived=> , 
	busy=> , 
	Error=> , 
	RxTimeout=> , 
	LenReceiveData=> , 
	RXbuffer:= gRxBuffer_TBP);

//testReal:=BYTE_TO_REAL(arr_RcvData_Temp);
//数据接收处理
recTon(IN:=RcvDataFlag, PT:=T#10MS);
IF recTon.Q THEN
	RcvDataFlag:=FALSE;
END_IF
reciveFtrig(CLK:=receive1.busy);
IF reciveFtrig.Q THEN
	arr_RcvDataByte:=arr_RcvDataByteTemp;
	arr_RcvDataByteTemp:=arr_RcvDataByteClear;
	RcvDataFlag:=TRUE;
	readDone:=TRUE;
	serialConnected:=TRUE;
	serialTimeoutError:=FALSE;
END_IF
againSendS3(IN:=NOT RcvDataFlag,PT:=T#5S);
IF againSendS3.Q THEN
	serialConnected:=FALSE;
	againSendS3(IN:=FALSE);
END_IF
ACT_Send();
ACT_LoopRead();
ACT_Reset();
ACT_Start();
ACT_Stop();

